LIN {X 0,Y 516.908,Z 331.095,A -85,B 0,C 180,E1 -5064.072,E2 -5064.072} C_VEL
LIN {X 0,Y 516.93,Z 331.097,A -85,B 0,C 180,E1 -5066.658,E2 -5066.658} C_VEL
LIN {X 0,Y 516.917,Z 331.093,A -85,B 0,C 180,E1 -5069.524,E2 -5069.524} C_VEL
LIN {X 0,Y 516.901,Z 331.095,A -85,B 0,C 180,E1 -5072.543,E2 -5072.543} C_VEL
LIN {X 0,Y 516.884,Z 331.1,A -85,B 0,C 180,E1 -5075.332,E2 -5075.332} C_VEL
LIN {X 0,Y 516.887,Z 331.098,A -85,B 0,C 180,E1 -5077.943,E2 -5077.943} C_VEL
LIN {X 0,Y 516.888,Z 331.102,A -85,B 0,C 180,E1 -5080.742,E2 -5080.742} C_VEL
LIN {X 0,Y 516.888,Z 331.102,A -85,B 0,C 180,E1 -5082.831,E2 -5082.831} C_VEL
LIN {X 0,Y 516.927,Z 331.093,A -85,B 0,C 180,E1 -5085.01,E2 -5085.01} C_VEL
LIN {X 0,Y 516.92,Z 331.096,A -85,B 0,C 180,E1 -5088.398,E2 -5088.398} C_VEL
LIN {X 0,Y 516.911,Z 331.249,A -85,B 0,C 180,E1 -5091.011,E2 -5091.011} C_VEL
LIN {X 0,Y 518.994,Z 341.632,A -85,B 0,C 180,E1 -5093.669,E2 -5093.669} C_VEL
LIN {X 0,Y 518.87,Z 348.689,A -85,B 0,C 180,E1 -5095.327,E2 -5095.327} C_VEL
LIN {X 0,Y 518.423,Z 362.259,A -85,B 0,C 180,E1 -5098.421,E2 -5098.421} C_VEL
LIN {X 0,Y 518.054,Z 376.981,A -85,B 0,C 180,E1 -5101.652,E2 -5101.652} C_VEL
LIN {X 0,Y 517.718,Z 390.09,A -85,B 0,C 180,E1 -5104.468,E2 -5104.468} C_VEL
LIN {X 0,Y 517.46,Z 402.865,A -85,B 0,C 180,E1 -5107.177,E2 -5107.177} C_VEL
LIN {X 0,Y 517.224,Z 417.474,A -85,B 0,C 180,E1 -5110.141,E2 -5110.141} C_VEL
LIN {X 0,Y 516.978,Z 432.958,A -85,B 0,C 180,E1 -5113.209,E2 -5113.209} C_VEL
LIN {X 0,Y 516.788,Z 447.169,A -85,B 0,C 180,E1 -5116.031,E2 -5116.031} C_VEL
LIN {X 0,Y 516.779,Z 447.609,A -85,B 0,C 180,E1 -5116.081,E2 -5116.081} C_VEL
LIN {X 0,Y 518.247,Z 458.294,A -85,B 0,C 180,E1 -5116.332,E2 -5116.332} C_VEL
LIN {X 0,Y 518.316,Z 465.73,A -85,B 0,C 180,E1 -5116.548,E2 -5116.548} C_VEL
LIN {X 0,Y 518.049,Z 479.168,A -85,B 0,C 180,E1 -5117.065,E2 -5117.065} C_VEL
LIN {X 0,Y 517.78,Z 490.854,A -85,B 0,C 180,E1 -5117.676,E2 -5117.676} C_VEL
LIN {X 0,Y 517.479,Z 502.323,A -85,B 0,C 180,E1 -5118.444,E2 -5118.444} C_VEL
LIN {X 0,Y 517.184,Z 512.955,A -85,B 0,C 180,E1 -5119.33,E2 -5119.33} C_VEL
LIN {X 0,Y 516.936,Z 521.664,A -85,B 0,C 180,E1 -5120.215,E2 -5120.215} C_VEL
LIN {X 0,Y 516.743,Z 529.713,A -85,B 0,C 180,E1 -5121.199,E2 -5121.199} C_VEL
LIN {X 0,Y 516.563,Z 537.593,A -85,B 0,C 180,E1 -5122.377,E2 -5122.377} C_VEL
LIN {X 0,Y 516.427,Z 544.854,A -85,B 0,C 180,E1 -5123.75,E2 -5123.75} C_VEL
LIN {X 0,Y 516.313,Z 549.687,A -85,B 0,C 180,E1 -5124.924,E2 -5124.924} C_VEL
LIN {X 0,Y 516.372,Z 553.401,A -85,B 0,C 180,E1 -5126.098,E2 -5126.098} C_VEL
LIN {X 0,Y 516.282,Z 555.3,A -85,B 0,C 180,E1 -5126.879,E2 -5126.879} C_VEL
LIN {X 0,Y 516.261,Z 556.732,A -85,B 0,C 180,E1 -5127.659,E2 -5127.659} C_VEL
LIN {X 0,Y 516.162,Z 558.365,A -85,B 0,C 180,E1 -5129.22,E2 -5129.22} C_VEL
LIN {X 0,Y 516.159,Z 558.585,A -85,B 0,C 180,E1 -5130,E2 -5130} C_VEL
LIN {X 0,Y 516.163,Z 558.362,A -85,B 0,C 180,E1 -5130.78,E2 -5130.78} C_VEL
LIN {X 0,Y 516.261,Z 556.725,A -85,B 0,C 180,E1 -5132.341,E2 -5132.341} C_VEL
LIN {X 0,Y 516.282,Z 555.285,A -85,B 0,C 180,E1 -5133.121,E2 -5133.121} C_VEL
LIN {X 0,Y 516.36,Z 552.268,A -85,B 0,C 180,E1 -5134.293,E2 -5134.293} C_VEL
LIN {X 0,Y 516.405,Z 548.17,A -85,B 0,C 180,E1 -5135.467,E2 -5135.467} C_VEL
LIN {X 0,Y 516.492,Z 541.976,A -85,B 0,C 180,E1 -5136.816,E2 -5136.816} C_VEL
LIN {X 0,Y 516.641,Z 534.976,A -85,B 0,C 180,E1 -5138.015,E2 -5138.015} C_VEL
LIN {X 0,Y 516.816,Z 526.424,A -85,B 0,C 180,E1 -5139.194,E2 -5139.194} C_VEL
LIN {X 0,Y 517.037,Z 517.651,A -85,B 0,C 180,E1 -5140.178,E2 -5140.178} C_VEL
LIN {X 0,Y 517.338,Z 506.848,A -85,B 0,C 180,E1 -5141.162,E2 -5141.162} C_VEL
LIN {X 0,Y 517.557,Z 495.523,A -85,B 0,C 180,E1 -5141.994,E2 -5141.994} C_VEL
LIN {X 0,Y 517.915,Z 483.454,A -85,B 0,C 180,E1 -5142.689,E2 -5142.689} C_VEL
LIN {X 0,Y 518.184,Z 469.779,A -85,B 0,C 180,E1 -5143.281,E2 -5143.281} C_VEL
LIN {X 0,Y 518.228,Z 458.613,A -85,B 0,C 180,E1 -5143.629,E2 -5143.629} C_VEL
LIN {X 0,Y 516.883,Z 448.292,A -85,B 0,C 180,E1 -5143.878,E2 -5143.878} C_VEL
LIN {X 0,Y 516.779,Z 446.249,A -85,B 0,C 180,E1 -5143.919,E2 -5143.919} C_VEL
LIN {X 0,Y 516.964,Z 430.116,A -85,B 0,C 180,E1 -5146.995,E2 -5146.995} C_VEL
LIN {X 0,Y 517.094,Z 415.047,A -85,B 0,C 180,E1 -5149.864,E2 -5149.864} C_VEL
LIN {X 0,Y 517.207,Z 399.793,A -85,B 0,C 180,E1 -5152.802,E2 -5152.802} C_VEL
LIN {X 0,Y 517.301,Z 385.694,A -85,B 0,C 180,E1 -5155.554,E2 -5155.554} C_VEL
LIN {X 0,Y 517.374,Z 371.54,A -85,B 0,C 180,E1 -5158.388,E2 -5158.388} C_VEL
LIN {X 0,Y 517.45,Z 358.184,A -85,B 0,C 180,E1 -5161.166,E2 -5161.166} C_VEL
LIN {X 0,Y 517.89,Z 341.975,A -85,B 0,C 180,E1 -5164.748,E2 -5164.748} C_VEL
LIN {X 0,Y 518.036,Z 337.974,A -85,B 0,C 180,E1 -5165.688,E2 -5165.688} C_VEL
LIN {X 0,Y 516.902,Z 331.103,A -85,B 0,C 180,E1 -5167.507,E2 -5167.507} C_VEL
LIN {X 0,Y 516.888,Z 331.103,A -85,B 0,C 180,E1 -5170.41,E2 -5170.41} C_VEL
LIN {X 0,Y 516.888,Z 331.102,A -85,B 0,C 180,E1 -5172.831,E2 -5172.831} C_VEL
LIN {X 0,Y 516.927,Z 331.095,A -85,B 0,C 180,E1 -5175.01,E2 -5175.01} C_VEL
LIN {X 0,Y 516.917,Z 331.097,A -85,B 0,C 180,E1 -5178.399,E2 -5178.399} C_VEL
LIN {X 0,Y 516.885,Z 331.101,A -85,B 0,C 180,E1 -5181.284,E2 -5181.284} C_VEL
LIN {X 0,Y 516.892,Z 331.101,A -85,B 0,C 180,E1 -5184.221,E2 -5184.221} C_VEL
LIN {X 0,Y 516.9,Z 331.1,A -85,B 0,C 180,E1 -5187.053,E2 -5187.053} C_VEL
LIN {X 0,Y 516.897,Z 331.101,A -85,B 0,C 180,E1 -5189.796,E2 -5189.796} C_VEL
LIN {X 0,Y 516.931,Z 331.095,A -85,B 0,C 180,E1 -5192.467,E2 -5192.467} C_VEL
LIN {X 0,Y 516.88,Z 331.1,A -85,B 0,C 180,E1 -5195.07,E2 -5195.07} C_VEL
LIN {X 0,Y 516.873,Z 331.102,A -85,B 0,C 180,E1 -5197.622,E2 -5197.622} C_VEL
LIN {X 0,Y 516.937,Z 331.096,A -85,B 0,C 180,E1 -5200.13,E2 -5200.13} C_VEL
LIN {X 0,Y 516.925,Z 331.098,A -85,B 0,C 180,E1 -5202.596,E2 -5202.596} C_VEL
LIN {X 0,Y 516.948,Z 331.094,A -85,B 0,C 180,E1 -5205.03,E2 -5205.03} C_VEL
LIN {X 0,Y 516.94,Z 331.279,A -85,B 0,C 180,E1 -5205.923,E2 -5205.923} C_VEL
LIN {X 0,Y 518.334,Z 336.946,A -85,B 0,C 180,E1 -5206.224,E2 -5206.224} C_VEL
LIN {X 0,Y 518.092,Z 348.48,A -85,B 0,C 180,E1 -5206.867,E2 -5206.867} C_VEL
LIN {X 0,Y 517.819,Z 359.058,A -85,B 0,C 180,E1 -5207.615,E2 -5207.615} C_VEL
LIN {X 0,Y 517.57,Z 368.563,A -85,B 0,C 180,E1 -5208.446,E2 -5208.446} C_VEL
LIN {X 0,Y 517.316,Z 377.754,A -85,B 0,C 180,E1 -5209.432,E2 -5209.432} C_VEL
LIN {X 0,Y 517.023,Z 386.607,A -85,B 0,C 180,E1 -5210.612,E2 -5210.612} C_VEL
LIN {X 0,Y 516.829,Z 393.689,A -85,B 0,C 180,E1 -5211.791,E2 -5211.791} C_VEL
LIN {X 0,Y 516.664,Z 399.315,A -85,B 0,C 180,E1 -5212.968,E2 -5212.968} C_VEL
LIN {X 0,Y 516.637,Z 403.722,A -85,B 0,C 180,E1 -5214.144,E2 -5214.144} C_VEL
LIN {X 0,Y 516.471,Z 407.079,A -85,B 0,C 180,E1 -5215.317,E2 -5215.317} C_VEL
LIN {X 0,Y 516.477,Z 408.761,A -85,B 0,C 180,E1 -5216.099,E2 -5216.099} C_VEL
LIN {X 0,Y 516.365,Z 410.885,A -85,B 0,C 180,E1 -5217.66,E2 -5217.66} C_VEL
LIN {X 0,Y 516.352,Z 411.375,A -85,B 0,C 180,E1 -5218.44,E2 -5218.44} C_VEL
LIN {X 0,Y 516.317,Z 411.149,A -85,B 0,C 180,E1 -5220,E2 -5220} C_VEL
LIN {X 0,Y 516.326,Z 410.458,A -85,B 0,C 180,E1 -5220.78,E2 -5220.78} C_VEL
LIN {X 0,Y 516.36,Z 409.365,A -85,B 0,C 180,E1 -5221.56,E2 -5221.56} C_VEL
LIN {X 0,Y 516.379,Z 407.875,A -85,B 0,C 180,E1 -5222.34,E2 -5222.34} C_VEL
LIN {X 0,Y 516.575,Z 404.822,A -85,B 0,C 180,E1 -5223.51,E2 -5223.51} C_VEL
LIN {X 0,Y 516.58,Z 400.77,A -85,B 0,C 180,E1 -5224.682,E2 -5224.682} C_VEL
LIN {X 0,Y 516.782,Z 394.527,A -85,B 0,C 180,E1 -5226.05,E2 -5226.05} C_VEL
LIN {X 0,Y 516.939,Z 387.732,A -85,B 0,C 180,E1 -5227.224,E2 -5227.224} C_VEL
LIN {X 0,Y 517.108,Z 379.256,A -85,B 0,C 180,E1 -5228.401,E2 -5228.401} C_VEL
LIN {X 0,Y 517.421,Z 370.5,A -85,B 0,C 180,E1 -5229.381,E2 -5229.381} C_VEL
LIN {X 0,Y 517.702,Z 360.917,A -85,B 0,C 180,E1 -5230.263,E2 -5230.263} C_VEL
LIN {X 0,Y 517.928,Z 350.396,A -85,B 0,C 180,E1 -5231.05,E2 -5231.05} C_VEL
LIN {X 0,Y 518.189,Z 338.681,A -85,B 0,C 180,E1 -5231.738,E2 -5231.738} C_VEL
LIN {X 0,Y 518.12,Z 335.637,A -85,B 0,C 180,E1 -5231.894,E2 -5231.894} C_VEL
LIN {X 0,Y 516.965,Z 331.093,A -85,B 0,C 180,E1 -5232.15,E2 -5232.15} C_VEL
LIN {X 0,Y 516.95,Z 331.092,A -85,B 0,C 180,E1 -5235.146,E2 -5235.146} C_VEL
LIN {X 0,Y 516.917,Z 331.092,A -85,B 0,C 180,E1 -5238.222,E2 -5238.222} C_VEL
LIN {X 0,Y 516.917,Z 331.097,A -85,B 0,C 180,E1 -5240.701,E2 -5240.701} C_VEL
LIN {X 0,Y 516.907,Z 331.098,A -85,B 0,C 180,E1 -5244.072,E2 -5244.072} C_VEL
LIN {X 0,Y 516.93,Z 331.094,A -85,B 0,C 180,E1 -5246.657,E2 -5246.657} C_VEL
LIN {X 0,Y 516.915,Z 331.099,A -85,B 0,C 180,E1 -5249.524,E2 -5249.524} C_VEL
LIN {X 0,Y 516.902,Z 331.095,A -85,B 0,C 180,E1 -5252.544,E2 -5252.544} C_VEL
LIN {X 0,Y 516.871,Z 331.101,A -85,B 0,C 180,E1 -5255.33,E2 -5255.33} C_VEL
LIN {X 0,Y 516.884,Z 331.097,A -85,B 0,C 180,E1 -5257.943,E2 -5257.943} C_VEL
LIN {X 0,Y 516.907,Z 331.097,A -85,B 0,C 180,E1 -5260.739,E2 -5260.739} C_VEL
LIN {X 0,Y 516.885,Z 331.102,A -85,B 0,C 180,E1 -5263.903,E2 -5263.903} C_VEL
LIN {X 0,Y 516.885,Z 331.099,A -85,B 0,C 180,E1 -5266.107,E2 -5266.107} C_VEL
LIN {X 0,Y 516.895,Z 331.096,A -85,B 0,C 180,E1 -5267.801,E2 -5267.801} C_VEL
LIN {X 0,Y 516.239,Z 331.179,A -85,B 0,C 180,E1 -5268.451,E2 -5268.451} C_VEL
LIN {X 0,Y 513.371,Z 331.538,A -85,B 0,C 180,E1 -5269.505,E2 -5269.505} C_VEL
LIN {X 0,Y 510.943,Z 331.839,A -85,B 0,C 180,E1 -5270.355,E2 -5270.355} C_VEL
LIN {X 0,Y 509.91,Z 331.971,A -85,B 0,C 180,E1 -5271.011,E2 -5271.011} C_VEL
LIN {X 0,Y 509.831,Z 331.975,A -85,B 0,C 180,E1 -5271.233,E2 -5271.233} C_VEL
LIN {X 0,Y 509.828,Z 331.981,A -85,B 0,C 180,E1 -5274.421,E2 -5274.421} C_VEL
LIN {X 0,Y 509.865,Z 331.973,A -85,B 0,C 180,E1 -5277.481,E2 -5277.481} C_VEL
LIN {X 0,Y 509.86,Z 331.975,A -85,B 0,C 180,E1 -5280.273,E2 -5280.273} C_VEL
LIN {X 0,Y 509.887,Z 331.972,A -85,B 0,C 180,E1 -5282.944,E2 -5282.944} C_VEL
LIN {X 0,Y 509.872,Z 331.973,A -85,B 0,C 180,E1 -5285.574,E2 -5285.574} C_VEL
LIN {X 0,Y 509.824,Z 331.978,A -85,B 0,C 180,E1 -5288.149,E2 -5288.149} C_VEL
LIN {X 0,Y 509.865,Z 331.974,A -85,B 0,C 180,E1 -5290.682,E2 -5290.682} C_VEL
LIN {X 0,Y 509.886,Z 331.968,A -85,B 0,C 180,E1 -5293.175,E2 -5293.175} C_VEL
LIN {X 0,Y 509.866,Z 331.976,A -85,B 0,C 180,E1 -5295.634,E2 -5295.634} C_VEL
LIN {X 0,Y 509.915,Z 331.968,A -85,B 0,C 180,E1 -5298.875,E2 -5298.875} C_VEL
LIN {X 0,Y 509.953,Z 331.961,A -85,B 0,C 180,E1 -5302.078,E2 -5302.078} C_VEL
LIN {X 0,Y 509.983,Z 331.963,A -85,B 0,C 180,E1 -5304.464,E2 -5304.464} C_VEL
LIN {X 0,Y 510.057,Z 331.949,A -85,B 0,C 180,E1 -5307.631,E2 -5307.631} C_VEL
LIN {X 0,Y 510.066,Z 331.946,A -85,B 0,C 180,E1 -5310.79,E2 -5310.79} C_VEL
LIN {X 0,Y 509.958,Z 331.963,A -85,B 0,C 180,E1 -5313.16,E2 -5313.16} C_VEL
LIN {X 0,Y 509.956,Z 331.961,A -85,B 0,C 180,E1 -5316.33,E2 -5316.33} C_VEL
LIN {X 0,Y 509.918,Z 331.969,A -85,B 0,C 180,E1 -5318.72,E2 -5318.72} C_VEL
LIN {X 0,Y 509.906,Z 331.97,A -85,B 0,C 180,E1 -5321.932,E2 -5321.932} C_VEL
LIN {X 0,Y 509.896,Z 331.968,A -85,B 0,C 180,E1 -5325.242,E2 -5325.242} C_VEL
LIN {X 0,Y 509.891,Z 331.97,A -85,B 0,C 180,E1 -5328.001,E2 -5328.001} C_VEL
LIN {X 0,Y 509.852,Z 331.977,A -85,B 0,C 180,E1 -5331.002,E2 -5331.002} C_VEL
LIN {X 0,Y 509.867,Z 331.976,A -85,B 0,C 180,E1 -5334.426,E2 -5334.426} C_VEL
LIN {X 0,Y 509.886,Z 331.97,A -85,B 0,C 180,E1 -5337.056,E2 -5337.056} C_VEL
LIN {X 0,Y 509.859,Z 331.977,A -85,B 0,C 180,E1 -5339.751,E2 -5339.751} C_VEL
LIN {X 0,Y 509.877,Z 331.97,A -85,B 0,C 180,E1 -5342.775,E2 -5342.775} C_VEL
LIN {X 0,Y 509.828,Z 331.979,A -85,B 0,C 180,E1 -5345.579,E2 -5345.579} C_VEL
LIN {X 0,Y 509.852,Z 331.975,A -85,B 0,C 180,E1 -5348.338,E2 -5348.338} C_VEL
LIN {X 0,Y 509.859,Z 331.973,A -85,B 0,C 180,E1 -5351.426,E2 -5351.426} C_VEL
LIN {X 0,Y 509.86,Z 331.974,A -85,B 0,C 180,E1 -5354.668,E2 -5354.668} C_VEL
LIN {X 0,Y 509.86,Z 331.974,A -85,B 0,C 180,E1 -5358.103,E2 -5358.103} C_VEL
LIN {X 0,Y 509.849,Z 331.974,A -85,B 0,C 180,E1 -5360.648,E2 -5360.648} C_VEL
LIN {X 0,Y 509.829,Z 331.976,A -85,B 0,C 180,E1 -5363.647,E2 -5363.647} C_VEL
LIN {X 0,Y 509.865,Z 331.977,A -85,B 0,C 180,E1 -5366.54,E2 -5366.54} C_VEL
LIN {X 0,Y 509.85,Z 331.974,A -85,B 0,C 180,E1 -5369.335,E2 -5369.335} C_VEL
LIN {X 0,Y 509.898,Z 331.972,A -85,B 0,C 180,E1 -5372.055,E2 -5372.055} C_VEL
LIN {X 0,Y 509.881,Z 331.97,A -85,B 0,C 180,E1 -5374.704,E2 -5374.704} C_VEL
LIN {X 0,Y 509.831,Z 331.978,A -85,B 0,C 180,E1 -5377.458,E2 -5377.458} C_VEL
LIN {X 0,Y 509.921,Z 331.963,A -85,B 0,C 180,E1 -5379.845,E2 -5379.845} C_VEL
LIN {X 0,Y 509.885,Z 331.969,A -85,B 0,C 180,E1 -5383.175,E2 -5383.175} C_VEL
LIN {X 0,Y 509.87,Z 331.974,A -85,B 0,C 180,E1 -5385.634,E2 -5385.634} C_VEL
LIN {X 0,Y 509.919,Z 331.966,A -85,B 0,C 180,E1 -5388.875,E2 -5388.875} C_VEL
LIN {X 0,Y 509.958,Z 331.96,A -85,B 0,C 180,E1 -5392.079,E2 -5392.079} C_VEL
LIN {X 0,Y 509.987,Z 331.959,A -85,B 0,C 180,E1 -5394.464,E2 -5394.464} C_VEL
LIN {X 0,Y 510.058,Z 331.946,A -85,B 0,C 180,E1 -5397.631,E2 -5397.631} C_VEL
LIN {X 0,Y 510.07,Z 331.947,A -85,B 0,C 180,E1 -5400.79,E2 -5400.79} C_VEL
LIN {X 0,Y 509.96,Z 331.961,A -85,B 0,C 180,E1 -5403.16,E2 -5403.16} C_VEL
LIN {X 0,Y 509.959,Z 331.961,A -85,B 0,C 180,E1 -5406.33,E2 -5406.33} C_VEL
LIN {X 0,Y 509.911,Z 331.97,A -85,B 0,C 180,E1 -5408.72,E2 -5408.72} C_VEL
LIN {X 0,Y 509.911,Z 331.966,A -85,B 0,C 180,E1 -5411.932,E2 -5411.932} C_VEL
LIN {X 0,Y 509.9,Z 331.966,A -85,B 0,C 180,E1 -5415.242,E2 -5415.242} C_VEL
LIN {X 0,Y 509.895,Z 331.973,A -85,B 0,C 180,E1 -5418.001,E2 -5418.001} C_VEL
LIN {X 0,Y 509.857,Z 331.975,A -85,B 0,C 180,E1 -5421.002,E2 -5421.002} C_VEL
LIN {X 0,Y 509.87,Z 331.973,A -85,B 0,C 180,E1 -5424.426,E2 -5424.426} C_VEL
LIN {X 0,Y 509.889,Z 331.972,A -85,B 0,C 180,E1 -5427.056,E2 -5427.056} C_VEL
LIN {X 0,Y 509.863,Z 331.973,A -85,B 0,C 180,E1 -5429.751,E2 -5429.751} C_VEL
LIN {X 0,Y 509.878,Z 331.969,A -85,B 0,C 180,E1 -5432.774,E2 -5432.774} C_VEL
LIN {X 0,Y 509.844,Z 331.98,A -85,B 0,C 180,E1 -5435.58,E2 -5435.58} C_VEL
LIN {X 0,Y 509.856,Z 331.973,A -85,B 0,C 180,E1 -5438.338,E2 -5438.338} C_VEL
LIN {X 0,Y 509.86,Z 331.974,A -85,B 0,C 180,E1 -5441.425,E2 -5441.425} C_VEL
LIN {X 0,Y 509.862,Z 331.977,A -85,B 0,C 180,E1 -5444.668,E2 -5444.668} C_VEL
LIN {X 0,Y 509.864,Z 331.977,A -85,B 0,C 180,E1 -5448.103,E2 -5448.103} C_VEL
LIN {X 0,Y 509.866,Z 332.045,A -85,B 0,C 180,E1 -5450.713,E2 -5450.713} C_VEL
LIN {X 0,Y 511.894,Z 342.129,A -85,B 0,C 180,E1 -5453.341,E2 -5453.341} C_VEL
LIN {X 0,Y 512.14,Z 346.602,A -85,B 0,C 180,E1 -5454.431,E2 -5454.431} C_VEL
LIN {X 0,Y 511.556,Z 361.233,A -85,B 0,C 180,E1 -5457.834,E2 -5457.834} C_VEL
LIN {X 0,Y 511.098,Z 376.354,A -85,B 0,C 180,E1 -5461.231,E2 -5461.231} C_VEL
LIN {X 0,Y 510.732,Z 389.473,A -85,B 0,C 180,E1 -5464.093,E2 -5464.093} C_VEL
LIN {X 0,Y 510.455,Z 402.496,A -85,B 0,C 180,E1 -5466.897,E2 -5466.897} C_VEL
LIN {X 0,Y 510.221,Z 414.988,A -85,B 0,C 180,E1 -5469.499,E2 -5469.499} C_VEL
LIN {X 0,Y 509.975,Z 431.227,A -85,B 0,C 180,E1 -5472.765,E2 -5472.765} C_VEL
LIN {X 0,Y 509.729,Z 445.315,A -85,B 0,C 180,E1 -5475.63,E2 -5475.63} C_VEL
LIN {X 0,Y 509.722,Z 446.55,A -85,B 0,C 180,E1 -5475.885,E2 -5475.885} C_VEL
LIN {X 0,Y 510.992,Z 457.207,A -85,B 0,C 180,E1 -5476.136,E2 -5476.136} C_VEL
LIN {X 0,Y 511.46,Z 462.268,A -85,B 0,C 180,E1 -5476.288,E2 -5476.288} C_VEL
LIN {X 0,Y 511.141,Z 474.694,A -85,B 0,C 180,E1 -5476.735,E2 -5476.735} C_VEL
LIN {X 0,Y 510.822,Z 487.491,A -85,B 0,C 180,E1 -5477.37,E2 -5477.37} C_VEL
LIN {X 0,Y 510.544,Z 498.597,A -85,B 0,C 180,E1 -5478.083,E2 -5478.083} C_VEL
LIN {X 0,Y 510.197,Z 509.748,A -85,B 0,C 180,E1 -5478.981,E2 -5478.981} C_VEL
LIN {X 0,Y 509.873,Z 520.644,A -85,B 0,C 180,E1 -5480.078,E2 -5480.078} C_VEL
LIN {X 0,Y 509.681,Z 528.707,A -85,B 0,C 180,E1 -5481.076,E2 -5481.076} C_VEL
LIN {X 0,Y 509.514,Z 536.607,A -85,B 0,C 180,E1 -5482.271,E2 -5482.271} C_VEL
LIN {X 0,Y 509.346,Z 543.872,A -85,B 0,C 180,E1 -5483.662,E2 -5483.662} C_VEL
LIN {X 0,Y 509.275,Z 548.715,A -85,B 0,C 180,E1 -5484.854,E2 -5484.854} C_VEL
LIN {X 0,Y 509.336,Z 552.432,A -85,B 0,C 180,E1 -5486.044,E2 -5486.044} C_VEL
LIN {X 0,Y 509.237,Z 554.326,A -85,B 0,C 180,E1 -5486.835,E2 -5486.835} C_VEL
LIN {X 0,Y 509.217,Z 555.758,A -85,B 0,C 180,E1 -5487.627,E2 -5487.627} C_VEL
LIN {X 0,Y 509.129,Z 557.385,A -85,B 0,C 180,E1 -5489.209,E2 -5489.209} C_VEL
LIN {X 0,Y 509.149,Z 557.596,A -85,B 0,C 180,E1 -5490,E2 -5490} C_VEL
LIN {X 0,Y 509.156,Z 557.366,A -85,B 0,C 180,E1 -5490.791,E2 -5490.791} C_VEL
LIN {X 0,Y 509.223,Z 555.705,A -85,B 0,C 180,E1 -5492.373,E2 -5492.373} C_VEL
LIN {X 0,Y 509.245,Z 554.244,A -85,B 0,C 180,E1 -5493.164,E2 -5493.164} C_VEL
LIN {X 0,Y 509.3,Z 551.196,A -85,B 0,C 180,E1 -5494.353,E2 -5494.353} C_VEL
LIN {X 0,Y 509.358,Z 547.068,A -85,B 0,C 180,E1 -5495.543,E2 -5495.543} C_VEL
LIN {X 0,Y 509.421,Z 541.059,A -85,B 0,C 180,E1 -5496.868,E2 -5496.868} C_VEL
LIN {X 0,Y 509.573,Z 533.79,A -85,B 0,C 180,E1 -5498.127,E2 -5498.127} C_VEL
LIN {X 0,Y 509.77,Z 525.183,A -85,B 0,C 180,E1 -5499.323,E2 -5499.323} C_VEL
LIN {X 0,Y 510.028,Z 515.354,A -85,B 0,C 180,E1 -5500.42,E2 -5500.42} C_VEL
LIN {X 0,Y 510.324,Z 504.283,A -85,B 0,C 180,E1 -5501.418,E2 -5501.418} C_VEL
LIN {X 0,Y 510.59,Z 492.953,A -85,B 0,C 180,E1 -5502.236,E2 -5502.236} C_VEL
LIN {X 0,Y 510.912,Z 480.946,A -85,B 0,C 180,E1 -5502.917,E2 -5502.917} C_VEL
LIN {X 0,Y 511.194,Z 468.245,A -85,B 0,C 180,E1 -5503.466,E2 -5503.466} C_VEL
LIN {X 0,Y 511.23,Z 459.231,A -85,B 0,C 180,E1 -5503.756,E2 -5503.756} C_VEL
LIN {X 0,Y 509.951,Z 448.798,A -85,B 0,C 180,E1 -5504.033,E2 -5504.033} C_VEL
LIN {X 0,Y 509.728,Z 444.968,A -85,B 0,C 180,E1 -5504.115,E2 -5504.115} C_VEL
LIN {X 0,Y 509.885,Z 428.825,A -85,B 0,C 180,E1 -5507.238,E2 -5507.238} C_VEL
LIN {X 0,Y 510.064,Z 412.232,A -85,B 0,C 180,E1 -5510.454,E2 -5510.454} C_VEL
LIN {X 0,Y 510.181,Z 395.371,A -85,B 0,C 180,E1 -5513.762,E2 -5513.762} C_VEL
LIN {X 0,Y 510.301,Z 380.687,A -85,B 0,C 180,E1 -5516.708,E2 -5516.708} C_VEL
LIN {X 0,Y 510.375,Z 365.654,A -85,B 0,C 180,E1 -5519.827,E2 -5519.827} C_VEL
LIN {X 0,Y 510.537,Z 353.484,A -85,B 0,C 180,E1 -5522.471,E2 -5522.471} C_VEL
LIN {X 0,Y 511.088,Z 340.285,A -85,B 0,C 180,E1 -5525.526,E2 -5525.526} C_VEL
LIN {X 0,Y 510.634,Z 336.003,A -85,B 0,C 180,E1 -5526.628,E2 -5526.628} C_VEL
LIN {X 0,Y 509.85,Z 331.981,A -85,B 0,C 180,E1 -5527.774,E2 -5527.774} C_VEL
LIN {X 0,Y 509.843,Z 331.979,A -85,B 0,C 180,E1 -5530.698,E2 -5530.698} C_VEL
LIN {X 0,Y 509.824,Z 331.981,A -85,B 0,C 180,E1 -5533.572,E2 -5533.572} C_VEL
LIN {X 0,Y 509.823,Z 331.979,A -85,B 0,C 180,E1 -5536.428,E2 -5536.428} C_VEL
LIN {X 0,Y 509.842,Z 331.977,A -85,B 0,C 180,E1 -5539.302,E2 -5539.302} C_VEL
LIN {X 0,Y 509.855,Z 331.976,A -85,B 0,C 180,E1 -5541.786,E2 -5541.786} C_VEL
LIN {X 0,Y 509.847,Z 331.978,A -85,B 0,C 180,E1 -5544.623,E2 -5544.623} C_VEL
LIN {X 0,Y 509.866,Z 331.975,A -85,B 0,C 180,E1 -5547.481,E2 -5547.481} C_VEL
LIN {X 0,Y 509.863,Z 331.975,A -85,B 0,C 180,E1 -5550.274,E2 -5550.274} C_VEL
LIN {X 0,Y 509.889,Z 331.973,A -85,B 0,C 180,E1 -5552.944,E2 -5552.944} C_VEL
LIN {X 0,Y 509.856,Z 331.978,A -85,B 0,C 180,E1 -5555.573,E2 -5555.573} C_VEL
LIN {X 0,Y 509.827,Z 331.982,A -85,B 0,C 180,E1 -5558.149,E2 -5558.149} C_VEL
LIN {X 0,Y 509.868,Z 331.976,A -85,B 0,C 180,E1 -5560.682,E2 -5560.682} C_VEL
LIN {X 0,Y 509.885,Z 331.973,A -85,B 0,C 180,E1 -5563.175,E2 -5563.175} C_VEL
LIN {X 0,Y 509.886,Z 332.091,A -85,B 0,C 180,E1 -5565.736,E2 -5565.736} C_VEL
LIN {X 0,Y 511.443,Z 338.53,A -85,B 0,C 180,E1 -5566.085,E2 -5566.085} C_VEL
LIN {X 0,Y 511.163,Z 350.716,A -85,B 0,C 180,E1 -5566.786,E2 -5566.786} C_VEL
LIN {X 0,Y 510.87,Z 362.015,A -85,B 0,C 180,E1 -5567.621,E2 -5567.621} C_VEL
LIN {X 0,Y 510.599,Z 371.402,A -85,B 0,C 180,E1 -5568.487,E2 -5568.487} C_VEL
LIN {X 0,Y 510.351,Z 380.243,A -85,B 0,C 180,E1 -5569.487,E2 -5569.487} C_VEL
LIN {X 0,Y 510.069,Z 388.834,A -85,B 0,C 180,E1 -5570.683,E2 -5570.683} C_VEL
LIN {X 0,Y 509.842,Z 395.671,A -85,B 0,C 180,E1 -5571.877,E2 -5571.877} C_VEL
LIN {X 0,Y 509.648,Z 401.468,A -85,B 0,C 180,E1 -5573.159,E2 -5573.159} C_VEL
LIN {X 0,Y 509.563,Z 405.95,A -85,B 0,C 180,E1 -5574.46,E2 -5574.46} C_VEL
LIN {X 0,Y 509.464,Z 408.083,A -85,B 0,C 180,E1 -5575.252,E2 -5575.252} C_VEL
LIN {X 0,Y 509.461,Z 409.77,A -85,B 0,C 180,E1 -5576.045,E2 -5576.045} C_VEL
LIN {X 0,Y 509.344,Z 411.897,A -85,B 0,C 180,E1 -5577.627,E2 -5577.627} C_VEL
LIN {X 0,Y 509.341,Z 412.386,A -85,B 0,C 180,E1 -5578.419,E2 -5578.419} C_VEL
LIN {X 0,Y 509.295,Z 412.157,A -85,B 0,C 180,E1 -5580,E2 -5580} C_VEL
LIN {X 0,Y 509.349,Z 410.365,A -85,B 0,C 180,E1 -5581.581,E2 -5581.581} C_VEL
LIN {X 0,Y 509.356,Z 408.871,A -85,B 0,C 180,E1 -5582.372,E2 -5582.372} C_VEL
LIN {X 0,Y 509.571,Z 405.805,A -85,B 0,C 180,E1 -5583.558,E2 -5583.558} C_VEL
LIN {X 0,Y 509.57,Z 401.739,A -85,B 0,C 180,E1 -5584.747,E2 -5584.747} C_VEL
LIN {X 0,Y 509.789,Z 395.475,A -85,B 0,C 180,E1 -5586.133,E2 -5586.133} C_VEL
LIN {X 0,Y 509.968,Z 388.665,A -85,B 0,C 180,E1 -5587.324,E2 -5587.324} C_VEL
LIN {X 0,Y 510.155,Z 380.169,A -85,B 0,C 180,E1 -5588.516,E2 -5588.516} C_VEL
LIN {X 0,Y 510.489,Z 371.4,A -85,B 0,C 180,E1 -5589.509,E2 -5589.509} C_VEL
LIN {X 0,Y 510.792,Z 361.804,A -85,B 0,C 180,E1 -5590.404,E2 -5590.404} C_VEL
LIN {X 0,Y 511.02,Z 351.287,A -85,B 0,C 180,E1 -5591.201,E2 -5591.201} C_VEL
LIN {X 0,Y 511.295,Z 339.58,A -85,B 0,C 180,E1 -5591.899,E2 -5591.899} C_VEL
LIN {X 0,Y 511.056,Z 336.268,A -85,B 0,C 180,E1 -5592.076,E2 -5592.076} C_VEL
LIN {X 0,Y 509.901,Z 331.972,A -85,B 0,C 180,E1 -5592.336,E2 -5592.336} C_VEL
LIN {X 0,Y 509.899,Z 331.971,A -85,B 0,C 180,E1 -5595.242,E2 -5595.242} C_VEL
LIN {X 0,Y 509.862,Z 331.971,A -85,B 0,C 180,E1 -5598.484,E2 -5598.484} C_VEL
LIN {X 0,Y 509.854,Z 331.978,A -85,B 0,C 180,E1 -5601.001,E2 -5601.001} C_VEL
LIN {X 0,Y 509.868,Z 331.976,A -85,B 0,C 180,E1 -5604.426,E2 -5604.426} C_VEL
LIN {X 0,Y 509.889,Z 331.969,A -85,B 0,C 180,E1 -5607.055,E2 -5607.055} C_VEL
LIN {X 0,Y 509.861,Z 331.977,A -85,B 0,C 180,E1 -5609.751,E2 -5609.751} C_VEL
LIN {X 0,Y 509.878,Z 331.971,A -85,B 0,C 180,E1 -5612.774,E2 -5612.774} C_VEL
LIN {X 0,Y 509.83,Z 331.976,A -85,B 0,C 180,E1 -5615.578,E2 -5615.578} C_VEL
LIN {X 0,Y 509.855,Z 331.976,A -85,B 0,C 180,E1 -5618.338,E2 -5618.338} C_VEL
LIN {X 0,Y 509.869,Z 331.972,A -85,B 0,C 180,E1 -5621.424,E2 -5621.424} C_VEL
LIN {X 0,Y 509.859,Z 331.973,A -85,B 0,C 180,E1 -5624.668,E2 -5624.668} C_VEL
LIN {X 0,Y 509.863,Z 331.973,A -85,B 0,C 180,E1 -5628.102,E2 -5628.102} C_VEL
LIN {X 0,Y 509.831,Z 331.975,A -85,B 0,C 180,E1 -5631.233,E2 -5631.233} C_VEL
LIN {X 0,Y 509.171,Z 332.058,A -85,B 0,C 180,E1 -5631.892,E2 -5631.892} C_VEL
LIN {X 0,Y 506.297,Z 332.419,A -85,B 0,C 180,E1 -5632.961,E2 -5632.961} C_VEL
LIN {X 0,Y 503.874,Z 332.719,A -85,B 0,C 180,E1 -5633.823,E2 -5633.823} C_VEL
LIN {X 0,Y 502.851,Z 332.851,A -85,B 0,C 180,E1 -5634.488,E2 -5634.488} C_VEL
LIN {X 0,Y 502.778,Z 332.854,A -85,B 0,C 180,E1 -5634.713,E2 -5634.713} C_VEL
LIN {X 0,Y 502.834,Z 332.848,A -85,B 0,C 180,E1 -5636.993,E2 -5636.993} C_VEL
LIN {X 0,Y 502.816,Z 332.854,A -85,B 0,C 180,E1 -5640.065,E2 -5640.065} C_VEL
LIN {X 0,Y 502.835,Z 332.848,A -85,B 0,C 180,E1 -5642.533,E2 -5642.533} C_VEL
LIN {X 0,Y 502.831,Z 332.852,A -85,B 0,C 180,E1 -5645.298,E2 -5645.298} C_VEL
LIN {X 0,Y 502.795,Z 332.852,A -85,B 0,C 180,E1 -5647.827,E2 -5647.827} C_VEL
LIN {X 0,Y 502.827,Z 332.855,A -85,B 0,C 180,E1 -5650.4,E2 -5650.4} C_VEL
LIN {X 0,Y 502.836,Z 332.847,A -85,B 0,C 180,E1 -5652.932,E2 -5652.932} C_VEL
LIN {X 0,Y 502.847,Z 332.849,A -85,B 0,C 180,E1 -5655.429,E2 -5655.429} C_VEL
LIN {X 0,Y 502.879,Z 332.844,A -85,B 0,C 180,E1 -5658.717,E2 -5658.717} C_VEL
LIN {X 0,Y 502.903,Z 332.84,A -85,B 0,C 180,E1 -5661.967,E2 -5661.967} C_VEL
LIN {X 0,Y 502.937,Z 332.84,A -85,B 0,C 180,E1 -5664.387,E2 -5664.387} C_VEL
LIN {X 0,Y 503.027,Z 332.824,A -85,B 0,C 180,E1 -5667.598,E2 -5667.598} C_VEL
LIN {X 0,Y 503.029,Z 332.828,A -85,B 0,C 180,E1 -5670,E2 -5670} C_VEL
LIN {X 0,Y 503.028,Z 332.824,A -85,B 0,C 180,E1 -5672.402,E2 -5672.402} C_VEL
LIN {X 0,Y 502.936,Z 332.838,A -85,B 0,C 180,E1 -5675.614,E2 -5675.614} C_VEL
LIN {X 0,Y 502.904,Z 332.84,A -85,B 0,C 180,E1 -5678.033,E2 -5678.033} C_VEL
LIN {X 0,Y 502.88,Z 332.842,A -85,B 0,C 180,E1 -5681.283,E2 -5681.283} C_VEL
LIN {X 0,Y 502.847,Z 332.846,A -85,B 0,C 180,E1 -5684.571,E2 -5684.571} C_VEL
LIN {X 0,Y 502.864,Z 332.846,A -85,B 0,C 180,E1 -5687.907,E2 -5687.907} C_VEL
LIN {X 0,Y 502.83,Z 332.849,A -85,B 0,C 180,E1 -5690.536,E2 -5690.536} C_VEL
LIN {X 0,Y 502.793,Z 332.858,A -85,B 0,C 180,E1 -5693.041,E2 -5693.041} C_VEL
LIN {X 0,Y 502.842,Z 332.847,A -85,B 0,C 180,E1 -5695.676,E2 -5695.676} C_VEL
LIN {X 0,Y 502.842,Z 332.85,A -85,B 0,C 180,E1 -5698.373,E2 -5698.373} C_VEL
LIN {X 0,Y 502.796,Z 332.856,A -85,B 0,C 180,E1 -5701.499,E2 -5701.499} C_VEL
LIN {X 0,Y 502.806,Z 332.851,A -85,B 0,C 180,E1 -5703.994,E2 -5703.994} C_VEL
LIN {X 0,Y 502.78,Z 332.86,A -85,B 0,C 180,E1 -5707.178,E2 -5707.178} C_VEL
LIN {X 0,Y 502.79,Z 332.854,A -85,B 0,C 180,E1 -5710.015,E2 -5710.015} C_VEL
LIN {X 0,Y 502.833,Z 332.852,A -85,B 0,C 180,E1 -5712.203,E2 -5712.203} C_VEL
LIN {X 0,Y 502.804,Z 332.854,A -85,B 0,C 180,E1 -5715.468,E2 -5715.468} C_VEL
LIN {X 0,Y 502.823,Z 332.85,A -85,B 0,C 180,E1 -5718.934,E2 -5718.934} C_VEL
LIN {X 0,Y 502.796,Z 332.851,A -85,B 0,C 180,E1 -5722.046,E2 -5722.046} C_VEL
LIN {X 0,Y 502.806,Z 332.855,A -85,B 0,C 180,E1 -5725.035,E2 -5725.035} C_VEL
LIN {X 0,Y 502.788,Z 332.856,A -85,B 0,C 180,E1 -5727.916,E2 -5727.916} C_VEL
LIN {X 0,Y 502.829,Z 332.85,A -85,B 0,C 180,E1 -5730.713,E2 -5730.713} C_VEL
LIN {X 0,Y 502.867,Z 332.849,A -85,B 0,C 180,E1 -5733.44,E2 -5733.44} C_VEL
LIN {X 0,Y 502.79,Z 332.853,A -85,B 0,C 180,E1 -5736.086,E2 -5736.086} C_VEL
LIN {X 0,Y 502.788,Z 332.857,A -85,B 0,C 180,E1 -5738.689,E2 -5738.689} C_VEL
LIN {X 0,Y 502.831,Z 332.848,A -85,B 0,C 180,E1 -5741.248,E2 -5741.248} C_VEL
LIN {X 0,Y 502.825,Z 332.85,A -85,B 0,C 180,E1 -5743.767,E2 -5743.767} C_VEL
LIN {X 0,Y 502.837,Z 332.852,A -85,B 0,C 180,E1 -5746.255,E2 -5746.255} C_VEL
LIN {X 0,Y 502.883,Z 332.842,A -85,B 0,C 180,E1 -5748.717,E2 -5748.717} C_VEL
LIN {X 0,Y 502.908,Z 332.839,A -85,B 0,C 180,E1 -5751.967,E2 -5751.967} C_VEL
LIN {X 0,Y 502.943,Z 332.836,A -85,B 0,C 180,E1 -5754.387,E2 -5754.387} C_VEL
LIN {X 0,Y 503.028,Z 332.822,A -85,B 0,C 180,E1 -5757.598,E2 -5757.598} C_VEL
LIN {X 0,Y 503.034,Z 332.826,A -85,B 0,C 180,E1 -5760,E2 -5760} C_VEL
LIN {X 0,Y 503.031,Z 332.825,A -85,B 0,C 180,E1 -5762.402,E2 -5762.402} C_VEL
LIN {X 0,Y 502.937,Z 332.839,A -85,B 0,C 180,E1 -5765.614,E2 -5765.614} C_VEL
LIN {X 0,Y 502.887,Z 332.842,A -85,B 0,C 180,E1 -5768.034,E2 -5768.034} C_VEL
LIN {X 0,Y 502.883,Z 332.843,A -85,B 0,C 180,E1 -5771.283,E2 -5771.283} C_VEL
LIN {X 0,Y 502.851,Z 332.848,A -85,B 0,C 180,E1 -5774.571,E2 -5774.571} C_VEL
LIN {X 0,Y 502.868,Z 332.849,A -85,B 0,C 180,E1 -5777.907,E2 -5777.907} C_VEL
LIN {X 0,Y 502.835,Z 332.848,A -85,B 0,C 180,E1 -5780.536,E2 -5780.536} C_VEL
LIN {X 0,Y 502.797,Z 332.856,A -85,B 0,C 180,E1 -5783.041,E2 -5783.041} C_VEL
LIN {X 0,Y 502.845,Z 332.847,A -85,B 0,C 180,E1 -5785.675,E2 -5785.675} C_VEL
LIN {X 0,Y 502.845,Z 332.852,A -85,B 0,C 180,E1 -5788.373,E2 -5788.373} C_VEL
LIN {X 0,Y 502.798,Z 332.852,A -85,B 0,C 180,E1 -5791.499,E2 -5791.499} C_VEL
LIN {X 0,Y 502.81,Z 332.851,A -85,B 0,C 180,E1 -5794.444,E2 -5794.444} C_VEL
LIN {X 0,Y 502.786,Z 332.857,A -85,B 0,C 180,E1 -5797.178,E2 -5797.178} C_VEL
LIN {X 0,Y 502.793,Z 332.853,A -85,B 0,C 180,E1 -5800.015,E2 -5800.015} C_VEL
LIN {X 0,Y 502.807,Z 332.854,A -85,B 0,C 180,E1 -5802.199,E2 -5802.199} C_VEL
LIN {X 0,Y 502.806,Z 332.852,A -85,B 0,C 180,E1 -5805.468,E2 -5805.468} C_VEL
LIN {X 0,Y 502.834,Z 332.852,A -85,B 0,C 180,E1 -5807.864,E2 -5807.864} C_VEL
LIN {X 0,Y 502.825,Z 333.026,A -85,B 0,C 180,E1 -5810.461,E2 -5810.461} C_VEL
LIN {X 0,Y 504.961,Z 343.532,A -85,B 0,C 180,E1 -5813.239,E2 -5813.239} C_VEL
LIN {X 0,Y 505.226,Z 347.589,A -85,B 0,C 180,E1 -5814.25,E2 -5814.25} C_VEL
LIN {X 0,Y 504.632,Z 360.686,A -85,B 0,C 180,E1 -5817.338,E2 -5817.338} C_VEL
LIN {X 0,Y 504.164,Z 373.742,A -85,B 0,C 180,E1 -5820.339,E2 -5820.339} C_VEL
LIN {X 0,Y 503.844,Z 387.854,A -85,B 0,C 180,E1 -5823.489,E2 -5823.489} C_VEL
LIN {X 0,Y 503.443,Z 401.886,A -85,B 0,C 180,E1 -5826.555,E2 -5826.555} C_VEL
LIN {X 0,Y 503.139,Z 416.038,A -85,B 0,C 180,E1 -5829.561,E2 -5829.561} C_VEL
LIN {X 0,Y 502.913,Z 431.546,A -85,B 0,C 180,E1 -5832.725,E2 -5832.725} C_VEL
LIN {X 0,Y 502.648,Z 445.682,A -85,B 0,C 180,E1 -5835.682,E2 -5835.682} C_VEL
LIN {X 0,Y 503.941,Z 457.493,A -85,B 0,C 180,E1 -5835.977,E2 -5835.977} C_VEL
LIN {X 0,Y 504.528,Z 462.007,A -85,B 0,C 180,E1 -5836.122,E2 -5836.122} C_VEL
LIN {X 0,Y 504.166,Z 474.76,A -85,B 0,C 180,E1 -5836.6,E2 -5836.6} C_VEL
LIN {X 0,Y 503.808,Z 486.643,A -85,B 0,C 180,E1 -5837.205,E2 -5837.205} C_VEL
LIN {X 0,Y 503.502,Z 498.931,A -85,B 0,C 180,E1 -5838.016,E2 -5838.016} C_VEL
LIN {X 0,Y 503.115,Z 509.807,A -85,B 0,C 180,E1 -5838.926,E2 -5838.926} C_VEL
LIN {X 0,Y 502.802,Z 519.622,A -85,B 0,C 180,E1 -5839.937,E2 -5839.937} C_VEL
LIN {X 0,Y 502.602,Z 527.698,A -85,B 0,C 180,E1 -5840.949,E2 -5840.949} C_VEL
LIN {X 0,Y 502.433,Z 535.615,A -85,B 0,C 180,E1 -5842.161,E2 -5842.161} C_VEL
LIN {X 0,Y 502.275,Z 542.889,A -85,B 0,C 180,E1 -5843.573,E2 -5843.573} C_VEL
LIN {X 0,Y 502.236,Z 547.741,A -85,B 0,C 180,E1 -5844.781,E2 -5844.781} C_VEL
LIN {X 0,Y 502.276,Z 551.458,A -85,B 0,C 180,E1 -5845.988,E2 -5845.988} C_VEL
LIN {X 0,Y 502.192,Z 553.352,A -85,B 0,C 180,E1 -5846.791,E2 -5846.791} C_VEL
LIN {X 0,Y 502.173,Z 554.784,A -85,B 0,C 180,E1 -5847.594,E2 -5847.594} C_VEL
LIN {X 0,Y 502.12,Z 555.793,A -85,B 0,C 180,E1 -5848.396,E2 -5848.396} C_VEL
LIN {X 0,Y 502.096,Z 556.401,A -85,B 0,C 180,E1 -5849.198,E2 -5849.198} C_VEL
LIN {X 0,Y 502.138,Z 556.608,A -85,B 0,C 180,E1 -5850,E2 -5850} C_VEL
LIN {X 0,Y 502.147,Z 556.371,A -85,B 0,C 180,E1 -5850.802,E2 -5850.802} C_VEL
LIN {X 0,Y 502.185,Z 554.68,A -85,B 0,C 180,E1 -5852.406,E2 -5852.406} C_VEL
LIN {X 0,Y 502.207,Z 553.202,A -85,B 0,C 180,E1 -5853.209,E2 -5853.209} C_VEL
LIN {X 0,Y 502.248,Z 550.125,A -85,B 0,C 180,E1 -5854.414,E2 -5854.414} C_VEL
LIN {X 0,Y 502.305,Z 545.966,A -85,B 0,C 180,E1 -5855.621,E2 -5855.621} C_VEL
LIN {X 0,Y 502.359,Z 539.675,A -85,B 0,C 180,E1 -5857.011,E2 -5857.011} C_VEL
LIN {X 0,Y 502.499,Z 532.599,A -85,B 0,C 180,E1 -5858.242,E2 -5858.242} C_VEL
LIN {X 0,Y 502.719,Z 523.939,A -85,B 0,C 180,E1 -5859.455,E2 -5859.455} C_VEL
LIN {X 0,Y 502.932,Z 514.045,A -85,B 0,C 180,E1 -5860.568,E2 -5860.568} C_VEL
LIN {X 0,Y 503.327,Z 502.929,A -85,B 0,C 180,E1 -5861.579,E2 -5861.579} C_VEL
LIN {X 0,Y 503.595,Z 491.678,A -85,B 0,C 180,E1 -5862.399,E2 -5862.399} C_VEL
LIN {X 0,Y 503.93,Z 479.464,A -85,B 0,C 180,E1 -5863.099,E2 -5863.099} C_VEL
LIN {X 0,Y 504.269,Z 466.723,A -85,B 0,C 180,E1 -5863.654,E2 -5863.654} C_VEL
LIN {X 0,Y 504.232,Z 459.901,A -85,B 0,C 180,E1 -5863.886,E2 -5863.886} C_VEL
LIN {X 0,Y 503.048,Z 449.786,A -85,B 0,C 180,E1 -5864.178,E2 -5864.178} C_VEL
LIN {X 0,Y 502.621,Z 443.675,A -85,B 0,C 180,E1 -5864.319,E2 -5864.319} C_VEL
LIN {X 0,Y 502.801,Z 429.654,A -85,B 0,C 180,E1 -5867.07,E2 -5867.07} C_VEL
LIN {X 0,Y 502.958,Z 413.604,A -85,B 0,C 180,E1 -5870.233,E2 -5870.233} C_VEL
LIN {X 0,Y 503.095,Z 397.411,A -85,B 0,C 180,E1 -5873.462,E2 -5873.462} C_VEL
LIN {X 0,Y 503.213,Z 383.364,A -85,B 0,C 180,E1 -5876.323,E2 -5876.323} C_VEL
LIN {X 0,Y 503.319,Z 369.421,A -85,B 0,C 180,E1 -5879.256,E2 -5879.256} C_VEL
LIN {X 0,Y 503.528,Z 356.786,A -85,B 0,C 180,E1 -5882.032,E2 -5882.032} C_VEL
LIN {X 0,Y 504.101,Z 342.64,A -85,B 0,C 180,E1 -5885.351,E2 -5885.351} C_VEL
LIN {X 0,Y 503.913,Z 338.571,A -85,B 0,C 180,E1 -5886.398,E2 -5886.398} C_VEL
LIN {X 0,Y 502.826,Z 332.856,A -85,B 0,C 180,E1 -5888.051,E2 -5888.051} C_VEL
LIN {X 0,Y 502.824,Z 332.853,A -85,B 0,C 180,E1 -5891.066,E2 -5891.066} C_VEL
LIN {X 0,Y 502.805,Z 332.857,A -85,B 0,C 180,E1 -5894.532,E2 -5894.532} C_VEL
LIN {X 0,Y 502.799,Z 332.854,A -85,B 0,C 180,E1 -5897.861,E2 -5897.861} C_VEL
LIN {X 0,Y 502.805,Z 332.853,A -85,B 0,C 180,E1 -5901.024,E2 -5901.024} C_VEL
LIN {X 0,Y 502.787,Z 332.858,A -85,B 0,C 180,E1 -5904.168,E2 -5904.168} C_VEL
LIN {X 0,Y 502.837,Z 332.852,A -85,B 0,C 180,E1 -5906.993,E2 -5906.993} C_VEL
LIN {X 0,Y 502.819,Z 332.853,A -85,B 0,C 180,E1 -5910.065,E2 -5910.065} C_VEL
LIN {X 0,Y 502.837,Z 332.851,A -85,B 0,C 180,E1 -5912.533,E2 -5912.533} C_VEL
LIN {X 0,Y 502.808,Z 332.855,A -85,B 0,C 180,E1 -5915.305,E2 -5915.305} C_VEL
LIN {X 0,Y 502.785,Z 332.857,A -85,B 0,C 180,E1 -5917.826,E2 -5917.826} C_VEL
LIN {X 0,Y 502.829,Z 332.852,A -85,B 0,C 180,E1 -5920.4,E2 -5920.4} C_VEL
LIN {X 0,Y 502.833,Z 332.852,A -85,B 0,C 180,E1 -5922.931,E2 -5922.931} C_VEL
LIN {X 0,Y 502.836,Z 332.943,A -85,B 0,C 180,E1 -5925.545,E2 -5925.545} C_VEL
LIN {X 0,Y 504.542,Z 339.126,A -85,B 0,C 180,E1 -5925.891,E2 -5925.891} C_VEL
LIN {X 0,Y 504.306,Z 351.408,A -85,B 0,C 180,E1 -5926.604,E2 -5926.604} C_VEL
LIN {X 0,Y 503.997,Z 362.856,A -85,B 0,C 180,E1 -5927.455,E2 -5927.455} C_VEL
LIN {X 0,Y 503.698,Z 372.247,A -85,B 0,C 180,E1 -5928.327,E2 -5928.327} C_VEL
LIN {X 0,Y 503.438,Z 381.125,A -85,B 0,C 180,E1 -5929.34,E2 -5929.34} C_VEL
LIN {X 0,Y 503.131,Z 389.751,A -85,B 0,C 180,E1 -5930.553,E2 -5930.553} C_VEL
LIN {X 0,Y 502.885,Z 396.63,A -85,B 0,C 180,E1 -5931.764,E2 -5931.764} C_VEL
LIN {X 0,Y 502.671,Z 402.441,A -85,B 0,C 180,E1 -5933.063,E2 -5933.063} C_VEL
LIN {X 0,Y 502.576,Z 406.94,A -85,B 0,C 180,E1 -5934.382,E2 -5934.382} C_VEL
LIN {X 0,Y 502.459,Z 409.087,A -85,B 0,C 180,E1 -5935.186,E2 -5935.186} C_VEL
LIN {X 0,Y 502.445,Z 410.778,A -85,B 0,C 180,E1 -5935.989,E2 -5935.989} C_VEL
LIN {X 0,Y 502.322,Z 412.909,A -85,B 0,C 180,E1 -5937.594,E2 -5937.594} C_VEL
LIN {X 0,Y 502.329,Z 413.396,A -85,B 0,C 180,E1 -5938.396,E2 -5938.396} C_VEL
LIN {X 0,Y 502.273,Z 413.162,A -85,B 0,C 180,E1 -5940,E2 -5940} C_VEL
LIN {X 0,Y 502.336,Z 411.365,A -85,B 0,C 180,E1 -5941.603,E2 -5941.603} C_VEL
LIN {X 0,Y 502.333,Z 409.866,A -85,B 0,C 180,E1 -5942.405,E2 -5942.405} C_VEL
LIN {X 0,Y 502.565,Z 406.787,A -85,B 0,C 180,E1 -5943.608,E2 -5943.608} C_VEL
LIN {X 0,Y 502.56,Z 402.705,A -85,B 0,C 180,E1 -5944.813,E2 -5944.813} C_VEL
LIN {X 0,Y 502.798,Z 396.422,A -85,B 0,C 180,E1 -5946.219,E2 -5946.219} C_VEL
LIN {X 0,Y 502.999,Z 389.598,A -85,B 0,C 180,E1 -5947.426,E2 -5947.426} C_VEL
LIN {X 0,Y 503.204,Z 381.081,A -85,B 0,C 180,E1 -5948.635,E2 -5948.635} C_VEL
LIN {X 0,Y 503.557,Z 372.301,A -85,B 0,C 180,E1 -5949.641,E2 -5949.641} C_VEL
LIN {X 0,Y 503.878,Z 362.692,A -85,B 0,C 180,E1 -5950.548,E2 -5950.548} C_VEL
LIN {X 0,Y 504.115,Z 352.227,A -85,B 0,C 180,E1 -5951.353,E2 -5951.353} C_VEL
LIN {X 0,Y 504.412,Z 340.473,A -85,B 0,C 180,E1 -5952.063,E2 -5952.063} C_VEL
LIN {X 0,Y 503.987,Z 337.03,A -85,B 0,C 180,E1 -5952.256,E2 -5952.256} C_VEL
LIN {X 0,Y 502.859,Z 332.848,A -85,B 0,C 180,E1 -5952.511,E2 -5952.511} C_VEL
LIN {X 0,Y 502.853,Z 332.85,A -85,B 0,C 180,E1 -5955.399,E2 -5955.399} C_VEL
LIN {X 0,Y 502.827,Z 332.85,A -85,B 0,C 180,E1 -5958.752,E2 -5958.752} C_VEL
LIN {X 0,Y 502.787,Z 332.855,A -85,B 0,C 180,E1 -5961.311,E2 -5961.311} C_VEL
LIN {X 0,Y 502.789,Z 332.855,A -85,B 0,C 180,E1 -5963.914,E2 -5963.914} C_VEL
LIN {X 0,Y 502.868,Z 332.846,A -85,B 0,C 180,E1 -5966.566,E2 -5966.566} C_VEL
LIN {X 0,Y 502.828,Z 332.851,A -85,B 0,C 180,E1 -5969.287,E2 -5969.287} C_VEL
LIN {X 0,Y 502.79,Z 332.854,A -85,B 0,C 180,E1 -5972.084,E2 -5972.084} C_VEL
LIN {X 0,Y 502.804,Z 332.857,A -85,B 0,C 180,E1 -5974.965,E2 -5974.965} C_VEL
LIN {X 0,Y 502.797,Z 332.852,A -85,B 0,C 180,E1 -5977.954,E2 -5977.954} C_VEL
LIN {X 0,Y 502.83,Z 332.849,A -85,B 0,C 180,E1 -5981.065,E2 -5981.065} C_VEL
LIN {X 0,Y 502.803,Z 332.853,A -85,B 0,C 180,E1 -5984.532,E2 -5984.532} C_VEL
LIN {X 0,Y 502.832,Z 332.85,A -85,B 0,C 180,E1 -5987.864,E2 -5987.864} C_VEL
LIN {X 0,Y 502.796,Z 332.854,A -85,B 0,C 180,E1 -5991.232,E2 -5991.232} C_VEL
LIN {X 0,Y 502.776,Z 332.856,A -85,B 0,C 180,E1 -5994.169,E2 -5994.169} C_VEL
LIN {X 0,Y 502.778,Z 332.854,A -85,B 0,C 180,E1 -5994.713,E2 -5994.713} C_VEL
LIN {X 0,Y 502.134,Z 332.936,A -85,B 0,C 180,E1 -5995.382,E2 -5995.382} C_VEL
LIN {X 0,Y 499.272,Z 333.296,A -85,B 0,C 180,E1 -5996.468,E2 -5996.468} C_VEL
LIN {X 0,Y 496.85,Z 333.594,A -85,B 0,C 180,E1 -5997.344,E2 -5997.344} C_VEL
LIN {X 0,Y 495.829,Z 333.725,A -85,B 0,C 180,E1 -5998.02,E2 -5998.02} C_VEL
LIN {X 0,Y 495.757,Z 333.733,A -85,B 0,C 180,E1 -5998.249,E2 -5998.249} C_VEL
LIN {X 0,Y 495.789,Z 333.729,A -85,B 0,C 180,E1 -6001.507,E2 -6001.507} C_VEL
LIN {X 0,Y 495.793,Z 333.726,A -85,B 0,C 180,E1 -6003.932,E2 -6003.932} C_VEL
LIN {X 0,Y 495.76,Z 333.732,A -85,B 0,C 180,E1 -6007.139,E2 -6007.139} C_VEL
LIN {X 0,Y 495.779,Z 333.729,A -85,B 0,C 180,E1 -6010.11,E2 -6010.11} C_VEL
LIN {X 0,Y 495.788,Z 333.726,A -85,B 0,C 180,E1 -6012.681,E2 -6012.681} C_VEL
LIN {X 0,Y 495.792,Z 333.726,A -85,B 0,C 180,E1 -6015.217,E2 -6015.217} C_VEL
LIN {X 0,Y 495.854,Z 333.718,A -85,B 0,C 180,E1 -6018.555,E2 -6018.555} C_VEL
LIN {X 0,Y 495.874,Z 333.715,A -85,B 0,C 180,E1 -6021.852,E2 -6021.852} C_VEL
LIN {X 0,Y 495.892,Z 333.716,A -85,B 0,C 180,E1 -6024.307,E2 -6024.307} C_VEL
LIN {X 0,Y 495.995,Z 333.7,A -85,B 0,C 180,E1 -6027.564,E2 -6027.564} C_VEL
LIN {X 0,Y 496.006,Z 333.697,A -85,B 0,C 180,E1 -6030.812,E2 -6030.812} C_VEL
LIN {X 0,Y 495.846,Z 333.721,A -85,B 0,C 180,E1 -6033.25,E2 -6033.25} C_VEL
LIN {X 0,Y 495.863,Z 333.718,A -85,B 0,C 180,E1 -6036.511,E2 -6036.511} C_VEL
LIN {X 0,Y 495.845,Z 333.722,A -85,B 0,C 180,E1 -6038.97,E2 -6038.97} C_VEL
LIN {X 0,Y 495.83,Z 333.724,A -85,B 0,C 180,E1 -6042.035,E2 -6042.035} C_VEL
LIN {X 0,Y 495.825,Z 333.722,A -85,B 0,C 180,E1 -6045.452,E2 -6045.452} C_VEL
LIN {X 0,Y 495.808,Z 333.723,A -85,B 0,C 180,E1 -6048.247,E2 -6048.247} C_VEL
LIN {X 0,Y 495.776,Z 333.729,A -85,B 0,C 180,E1 -6050.757,E2 -6050.757} C_VEL
LIN {X 0,Y 495.75,Z 333.732,A -85,B 0,C 180,E1 -6053.387,E2 -6053.387} C_VEL
LIN {X 0,Y 495.793,Z 333.728,A -85,B 0,C 180,E1 -6056.068,E2 -6056.068} C_VEL
LIN {X 0,Y 495.774,Z 333.728,A -85,B 0,C 180,E1 -6058.815,E2 -6058.815} C_VEL
LIN {X 0,Y 495.759,Z 333.734,A -85,B 0,C 180,E1 -6061.726,E2 -6061.726} C_VEL
LIN {X 0,Y 495.771,Z 333.727,A -85,B 0,C 180,E1 -6064.694,E2 -6064.694} C_VEL
LIN {X 0,Y 495.731,Z 333.734,A -85,B 0,C 180,E1 -6067.562,E2 -6067.562} C_VEL
LIN {X 0,Y 495.769,Z 333.732,A -85,B 0,C 180,E1 -6070.7,E2 -6070.7} C_VEL
LIN {X 0,Y 495.738,Z 333.734,A -85,B 0,C 180,E1 -6073.696,E2 -6073.696} C_VEL
LIN {X 0,Y 495.732,Z 333.735,A -85,B 0,C 180,E1 -6076.306,E2 -6076.306} C_VEL
LIN {X 0,Y 495.77,Z 333.733,A -85,B 0,C 180,E1 -6079.3,E2 -6079.3} C_VEL
LIN {X 0,Y 495.733,Z 333.732,A -85,B 0,C 180,E1 -6082.439,E2 -6082.439} C_VEL
LIN {X 0,Y 495.785,Z 333.726,A -85,B 0,C 180,E1 -6085.457,E2 -6085.457} C_VEL
LIN {X 0,Y 495.76,Z 333.733,A -85,B 0,C 180,E1 -6088.364,E2 -6088.364} C_VEL
LIN {X 0,Y 495.792,Z 333.729,A -85,B 0,C 180,E1 -6091.507,E2 -6091.507} C_VEL
LIN {X 0,Y 495.796,Z 333.727,A -85,B 0,C 180,E1 -6093.933,E2 -6093.933} C_VEL
LIN {X 0,Y 495.765,Z 333.734,A -85,B 0,C 180,E1 -6097.14,E2 -6097.14} C_VEL
LIN {X 0,Y 495.774,Z 333.727,A -85,B 0,C 180,E1 -6100.11,E2 -6100.11} C_VEL
LIN {X 0,Y 495.785,Z 333.73,A -85,B 0,C 180,E1 -6102.681,E2 -6102.681} C_VEL
LIN {X 0,Y 495.796,Z 333.725,A -85,B 0,C 180,E1 -6105.217,E2 -6105.217} C_VEL
LIN {X 0,Y 495.857,Z 333.718,A -85,B 0,C 180,E1 -6108.555,E2 -6108.555} C_VEL
LIN {X 0,Y 495.879,Z 333.715,A -85,B 0,C 180,E1 -6111.852,E2 -6111.852} C_VEL
LIN {X 0,Y 495.901,Z 333.712,A -85,B 0,C 180,E1 -6114.307,E2 -6114.307} C_VEL
LIN {X 0,Y 495.997,Z 333.698,A -85,B 0,C 180,E1 -6117.564,E2 -6117.564} C_VEL
LIN {X 0,Y 496.011,Z 333.698,A -85,B 0,C 180,E1 -6120.812,E2 -6120.812} C_VEL
LIN {X 0,Y 495.847,Z 333.72,A -85,B 0,C 180,E1 -6123.25,E2 -6123.25} C_VEL
LIN {X 0,Y 495.866,Z 333.717,A -85,B 0,C 180,E1 -6126.511,E2 -6126.511} C_VEL
LIN {X 0,Y 495.841,Z 333.723,A -85,B 0,C 180,E1 -6128.97,E2 -6128.97} C_VEL
LIN {X 0,Y 495.834,Z 333.721,A -85,B 0,C 180,E1 -6132.035,E2 -6132.035} C_VEL
LIN {X 0,Y 495.83,Z 333.719,A -85,B 0,C 180,E1 -6135.452,E2 -6135.452} C_VEL
LIN {X 0,Y 495.813,Z 333.725,A -85,B 0,C 180,E1 -6138.247,E2 -6138.247} C_VEL
LIN {X 0,Y 495.78,Z 333.727,A -85,B 0,C 180,E1 -6140.756,E2 -6140.756} C_VEL
LIN {X 0,Y 495.753,Z 333.734,A -85,B 0,C 180,E1 -6143.387,E2 -6143.387} C_VEL
LIN {X 0,Y 495.796,Z 333.726,A -85,B 0,C 180,E1 -6146.068,E2 -6146.068} C_VEL
LIN {X 0,Y 495.777,Z 333.729,A -85,B 0,C 180,E1 -6148.815,E2 -6148.815} C_VEL
LIN {X 0,Y 495.76,Z 333.731,A -85,B 0,C 180,E1 -6151.725,E2 -6151.725} C_VEL
LIN {X 0,Y 495.78,Z 333.726,A -85,B 0,C 180,E1 -6154.695,E2 -6154.695} C_VEL
LIN {X 0,Y 495.736,Z 333.736,A -85,B 0,C 180,E1 -6157.561,E2 -6157.561} C_VEL
LIN {X 0,Y 495.771,Z 333.731,A -85,B 0,C 180,E1 -6160.7,E2 -6160.7} C_VEL
LIN {X 0,Y 495.739,Z 333.734,A -85,B 0,C 180,E1 -6164.001,E2 -6164.001} C_VEL
LIN {X 0,Y 495.738,Z 333.733,A -85,B 0,C 180,E1 -6167.118,E2 -6167.118} C_VEL
LIN {X 0,Y 495.766,Z 333.823,A -85,B 0,C 180,E1 -6170.158,E2 -6170.158} C_VEL
LIN {X 0,Y 498.002,Z 344.853,A -85,B 0,C 180,E1 -6173.12,E2 -6173.12} C_VEL
LIN {X 0,Y 498.319,Z 349.031,A -85,B 0,C 180,E1 -6174.176,E2 -6174.176} C_VEL
LIN {X 0,Y 497.696,Z 362.099,A -85,B 0,C 180,E1 -6177.307,E2 -6177.307} C_VEL
LIN {X 0,Y 497.181,Z 375.155,A -85,B 0,C 180,E1 -6180.346,E2 -6180.346} C_VEL
LIN {X 0,Y 496.81,Z 389.221,A -85,B 0,C 180,E1 -6183.538,E2 -6183.538} C_VEL
LIN {X 0,Y 496.393,Z 403.276,A -85,B 0,C 180,E1 -6186.645,E2 -6186.645} C_VEL
LIN {X 0,Y 496.06,Z 417.397,A -85,B 0,C 180,E1 -6189.689,E2 -6189.689} C_VEL
LIN {X 0,Y 495.847,Z 431.666,A -85,B 0,C 180,E1 -6192.683,E2 -6192.683} C_VEL
LIN {X 0,Y 495.577,Z 444.815,A -85,B 0,C 180,E1 -6195.473,E2 -6195.473} C_VEL
LIN {X 0,Y 497.046,Z 458.644,A -85,B 0,C 180,E1 -6195.843,E2 -6195.843} C_VEL
LIN {X 0,Y 497.516,Z 463.229,A -85,B 0,C 180,E1 -6196,E2 -6196} C_VEL
LIN {X 0,Y 497.144,Z 475.903,A -85,B 0,C 180,E1 -6196.511,E2 -6196.511} C_VEL
LIN {X 0,Y 496.775,Z 487.676,A -85,B 0,C 180,E1 -6197.146,E2 -6197.146} C_VEL
LIN {X 0,Y 496.458,Z 499.203,A -85,B 0,C 180,E1 -6197.948,E2 -6197.948} C_VEL
LIN {X 0,Y 496.033,Z 509.853,A -85,B 0,C 180,E1 -6198.869,E2 -6198.869} C_VEL
LIN {X 0,Y 495.76,Z 518.604,A -85,B 0,C 180,E1 -6199.793,E2 -6199.793} C_VEL
LIN {X 0,Y 495.529,Z 526.69,A -85,B 0,C 180,E1 -6200.819,E2 -6200.819} C_VEL
LIN {X 0,Y 495.376,Z 534.627,A -85,B 0,C 180,E1 -6202.049,E2 -6202.049} C_VEL
LIN {X 0,Y 495.213,Z 541.906,A -85,B 0,C 180,E1 -6203.481,E2 -6203.481} C_VEL
LIN {X 0,Y 495.176,Z 546.764,A -85,B 0,C 180,E1 -6204.707,E2 -6204.707} C_VEL
LIN {X 0,Y 495.217,Z 550.482,A -85,B 0,C 180,E1 -6205.931,E2 -6205.931} C_VEL
LIN {X 0,Y 495.145,Z 552.378,A -85,B 0,C 180,E1 -6206.745,E2 -6206.745} C_VEL
LIN {X 0,Y 495.129,Z 553.81,A -85,B 0,C 180,E1 -6207.559,E2 -6207.559} C_VEL
LIN {X 0,Y 495.083,Z 554.817,A -85,B 0,C 180,E1 -6208.373,E2 -6208.373} C_VEL
LIN {X 0,Y 495.125,Z 555.619,A -85,B 0,C 180,E1 -6210,E2 -6210} C_VEL
LIN {X 0,Y 495.136,Z 555.375,A -85,B 0,C 180,E1 -6210.813,E2 -6210.813} C_VEL
LIN {X 0,Y 495.096,Z 554.716,A -85,B 0,C 180,E1 -6211.627,E2 -6211.627} C_VEL
LIN {X 0,Y 495.147,Z 553.651,A -85,B 0,C 180,E1 -6212.44,E2 -6212.44} C_VEL
LIN {X 0,Y 495.169,Z 552.16,A -85,B 0,C 180,E1 -6213.255,E2 -6213.255} C_VEL
LIN {X 0,Y 495.202,Z 549.056,A -85,B 0,C 180,E1 -6214.477,E2 -6214.477} C_VEL
LIN {X 0,Y 495.25,Z 544.863,A -85,B 0,C 180,E1 -6215.701,E2 -6215.701} C_VEL
LIN {X 0,Y 495.317,Z 538.533,A -85,B 0,C 180,E1 -6217.111,E2 -6217.111} C_VEL
LIN {X 0,Y 495.455,Z 531.402,A -85,B 0,C 180,E1 -6218.36,E2 -6218.36} C_VEL
LIN {X 0,Y 495.634,Z 522.687,A -85,B 0,C 180,E1 -6219.591,E2 -6219.591} C_VEL
LIN {X 0,Y 495.902,Z 512.742,A -85,B 0,C 180,E1 -6220.72,E2 -6220.72} C_VEL
LIN {X 0,Y 496.326,Z 501.574,A -85,B 0,C 180,E1 -6221.745,E2 -6221.745} C_VEL
LIN {X 0,Y 496.581,Z 490.875,A -85,B 0,C 180,E1 -6222.537,E2 -6222.537} C_VEL
LIN {X 0,Y 496.946,Z 477.981,A -85,B 0,C 180,E1 -6223.286,E2 -6223.286} C_VEL
LIN {X 0,Y 497.336,Z 465.191,A -85,B 0,C 180,E1 -6223.848,E2 -6223.848} C_VEL
LIN {X 0,Y 497.204,Z 460.323,A -85,B 0,C 180,E1 -6224.021,E2 -6224.021} C_VEL
LIN {X 0,Y 496.103,Z 450.33,A -85,B 0,C 180,E1 -6224.328,E2 -6224.328} C_VEL
LIN {X 0,Y 495.566,Z 442.391,A -85,B 0,C 180,E1 -6224.527,E2 -6224.527} C_VEL
LIN {X 0,Y 495.758,Z 426.262,A -85,B 0,C 180,E1 -6227.746,E2 -6227.746} C_VEL
LIN {X 0,Y 495.906,Z 410.209,A -85,B 0,C 180,E1 -6230.968,E2 -6230.968} C_VEL
LIN {X 0,Y 496.044,Z 395.154,A -85,B 0,C 180,E1 -6234.038,E2 -6234.038} C_VEL
LIN {X 0,Y 496.21,Z 380.124,A -85,B 0,C 180,E1 -6237.179,E2 -6237.179} C_VEL
LIN {X 0,Y 496.371,Z 365.921,A -85,B 0,C 180,E1 -6240.267,E2 -6240.267} C_VEL
LIN {X 0,Y 496.597,Z 354.126,A -85,B 0,C 180,E1 -6242.965,E2 -6242.965} C_VEL
LIN {X 0,Y 497.223,Z 342.321,A -85,B 0,C 180,E1 -6245.851,E2 -6245.851} C_VEL
LIN {X 0,Y 496.265,Z 336.355,A -85,B 0,C 180,E1 -6247.527,E2 -6247.527} C_VEL
LIN {X 0,Y 495.783,Z 333.733,A -85,B 0,C 180,E1 -6248.329,E2 -6248.329} C_VEL
LIN {X 0,Y 495.76,Z 333.734,A -85,B 0,C 180,E1 -6251.293,E2 -6251.293} C_VEL
LIN {X 0,Y 495.738,Z 333.736,A -85,B 0,C 180,E1 -6254.001,E2 -6254.001} C_VEL
LIN {X 0,Y 495.73,Z 333.737,A -85,B 0,C 180,E1 -6257.117,E2 -6257.117} C_VEL
LIN {X 0,Y 495.762,Z 333.733,A -85,B 0,C 180,E1 -6259.953,E2 -6259.953} C_VEL
LIN {X 0,Y 495.734,Z 333.734,A -85,B 0,C 180,E1 -6262.553,E2 -6262.553} C_VEL
LIN {X 0,Y 495.788,Z 333.729,A -85,B 0,C 180,E1 -6265.457,E2 -6265.457} C_VEL
LIN {X 0,Y 495.76,Z 333.734,A -85,B 0,C 180,E1 -6268.364,E2 -6268.364} C_VEL
LIN {X 0,Y 495.792,Z 333.728,A -85,B 0,C 180,E1 -6271.507,E2 -6271.507} C_VEL
LIN {X 0,Y 495.785,Z 333.729,A -85,B 0,C 180,E1 -6273.932,E2 -6273.932} C_VEL
LIN {X 0,Y 495.764,Z 333.734,A -85,B 0,C 180,E1 -6277.14,E2 -6277.14} C_VEL
LIN {X 0,Y 495.776,Z 333.732,A -85,B 0,C 180,E1 -6280.11,E2 -6280.11} C_VEL
LIN {X 0,Y 495.786,Z 333.732,A -85,B 0,C 180,E1 -6282.681,E2 -6282.681} C_VEL
LIN {X 0,Y 495.826,Z 333.915,A -85,B 0,C 180,E1 -6285.349,E2 -6285.349} C_VEL
LIN {X 0,Y 497.739,Z 341.789,A -85,B 0,C 180,E1 -6285.798,E2 -6285.798} C_VEL
LIN {X 0,Y 497.419,Z 353.725,A -85,B 0,C 180,E1 -6286.519,E2 -6286.519} C_VEL
LIN {X 0,Y 497.12,Z 363.797,A -85,B 0,C 180,E1 -6287.288,E2 -6287.288} C_VEL
LIN {X 0,Y 496.807,Z 373.118,A -85,B 0,C 180,E1 -6288.163,E2 -6288.163} C_VEL
LIN {X 0,Y 496.53,Z 382.017,A -85,B 0,C 180,E1 -6289.19,E2 -6289.19} C_VEL
LIN {X 0,Y 496.195,Z 390.666,A -85,B 0,C 180,E1 -6290.42,E2 -6290.42} C_VEL
LIN {X 0,Y 495.931,Z 397.589,A -85,B 0,C 180,E1 -6291.648,E2 -6291.648} C_VEL
LIN {X 0,Y 495.696,Z 403.415,A -85,B 0,C 180,E1 -6292.965,E2 -6292.965} C_VEL
LIN {X 0,Y 495.59,Z 407.931,A -85,B 0,C 180,E1 -6294.303,E2 -6294.303} C_VEL
LIN {X 0,Y 495.456,Z 410.091,A -85,B 0,C 180,E1 -6295.118,E2 -6295.118} C_VEL
LIN {X 0,Y 495.43,Z 411.787,A -85,B 0,C 180,E1 -6295.933,E2 -6295.933} C_VEL
LIN {X 0,Y 495.3,Z 413.921,A -85,B 0,C 180,E1 -6297.56,E2 -6297.56} C_VEL
LIN {X 0,Y 495.315,Z 414.407,A -85,B 0,C 180,E1 -6298.374,E2 -6298.374} C_VEL
LIN {X 0,Y 495.264,Z 414.489,A -85,B 0,C 180,E1 -6299.187,E2 -6299.187} C_VEL
LIN {X 0,Y 495.268,Z 413.459,A -85,B 0,C 180,E1 -6300.813,E2 -6300.813} C_VEL
LIN {X 0,Y 495.322,Z 412.364,A -85,B 0,C 180,E1 -6301.626,E2 -6301.626} C_VEL
LIN {X 0,Y 495.31,Z 410.856,A -85,B 0,C 180,E1 -6302.44,E2 -6302.44} C_VEL
LIN {X 0,Y 495.557,Z 407.764,A -85,B 0,C 180,E1 -6303.659,E2 -6303.659} C_VEL
LIN {X 0,Y 495.551,Z 403.668,A -85,B 0,C 180,E1 -6304.881,E2 -6304.881} C_VEL
LIN {X 0,Y 495.81,Z 397.368,A -85,B 0,C 180,E1 -6306.307,E2 -6306.307} C_VEL
LIN {X 0,Y 496.031,Z 390.531,A -85,B 0,C 180,E1 -6307.531,E2 -6307.531} C_VEL
LIN {X 0,Y 496.257,Z 381.993,A -85,B 0,C 180,E1 -6308.757,E2 -6308.757} C_VEL
LIN {X 0,Y 496.627,Z 373.203,A -85,B 0,C 180,E1 -6309.777,E2 -6309.777} C_VEL
LIN {X 0,Y 497.004,Z 362.409,A -85,B 0,C 180,E1 -6310.799,E2 -6310.799} C_VEL
LIN {X 0,Y 497.273,Z 351.785,A -85,B 0,C 180,E1 -6311.602,E2 -6311.602} C_VEL
LIN {X 0,Y 497.553,Z 340.299,A -85,B 0,C 180,E1 -6312.289,E2 -6312.289} C_VEL
LIN {X 0,Y 495.82,Z 333.724,A -85,B 0,C 180,E1 -6312.686,E2 -6312.686} C_VEL
LIN {X 0,Y 495.811,Z 333.727,A -85,B 0,C 180,E1 -6315.624,E2 -6315.624} C_VEL
LIN {X 0,Y 495.783,Z 333.731,A -85,B 0,C 180,E1 -6319.028,E2 -6319.028} C_VEL
LIN {X 0,Y 495.747,Z 333.731,A -85,B 0,C 180,E1 -6321.629,E2 -6321.629} C_VEL
LIN {X 0,Y 495.782,Z 333.728,A -85,B 0,C 180,E1 -6324.873,E2 -6324.873} C_VEL
LIN {X 0,Y 495.818,Z 333.723,A -85,B 0,C 180,E1 -6326.974,E2 -6326.974} C_VEL
LIN {X 0,Y 495.769,Z 333.73,A -85,B 0,C 180,E1 -6330.147,E2 -6330.147} C_VEL
LIN {X 0,Y 495.796,Z 333.729,A -85,B 0,C 180,E1 -6333.244,E2 -6333.244} C_VEL
LIN {X 0,Y 495.723,Z 333.732,A -85,B 0,C 180,E1 -6336.088,E2 -6336.088} C_VEL
LIN {X 0,Y 495.772,Z 333.732,A -85,B 0,C 180,E1 -6338.769,E2 -6338.769} C_VEL
LIN {X 0,Y 495.764,Z 333.732,A -85,B 0,C 180,E1 -6341.78,E2 -6341.78} C_VEL
LIN {X 0,Y 495.752,Z 333.732,A -85,B 0,C 180,E1 -6345.139,E2 -6345.139} C_VEL
LIN {X 0,Y 495.78,Z 333.727,A -85,B 0,C 180,E1 -6348.221,E2 -6348.221} C_VEL
LIN {X 0,Y 495.752,Z 333.731,A -85,B 0,C 180,E1 -6351.408,E2 -6351.408} C_VEL
LIN {X 0,Y 495.745,Z 333.733,A -85,B 0,C 180,E1 -6354.713,E2 -6354.713} C_VEL
LIN {X 0,Y 495.77,Z 333.728,A -85,B 0,C 180,E1 -6357.406,E2 -6357.406} C_VEL
LIN {X 0,Y 495.757,Z 333.733,A -85,B 0,C 180,E1 -6358.249,E2 -6358.249} C_VEL
LIN {X 0,Y 495.124,Z 333.818,A -85,B 0,C 180,E1 -6358.927,E2 -6358.927} C_VEL
LIN {X 0,Y 492.296,Z 334.174,A -85,B 0,C 180,E1 -6360.028,E2 -6360.028} C_VEL
LIN {X 0,Y 489.878,Z 334.471,A -85,B 0,C 180,E1 -6360.915,E2 -6360.915} C_VEL
LIN {X 0,Y 488.828,Z 334.597,A -85,B 0,C 180,E1 -6361.6,E2 -6361.6} C_VEL
LIN {X 0,Y 488.737,Z 334.606,A -85,B 0,C 180,E1 -6361.832,E2 -6361.832} C_VEL
LIN {X 0,Y 488.749,Z 334.603,A -85,B 0,C 180,E1 -6364.444,E2 -6364.444} C_VEL
LIN {X 0,Y 488.723,Z 334.608,A -85,B 0,C 180,E1 -6367.153,E2 -6367.153} C_VEL
LIN {X 0,Y 488.73,Z 334.605,A -85,B 0,C 180,E1 -6369.811,E2 -6369.811} C_VEL
LIN {X 0,Y 488.736,Z 334.607,A -85,B 0,C 180,E1 -6372.423,E2 -6372.423} C_VEL
LIN {X 0,Y 488.764,Z 334.601,A -85,B 0,C 180,E1 -6375,E2 -6375} C_VEL
LIN {X 0,Y 488.807,Z 334.596,A -85,B 0,C 180,E1 -6378.388,E2 -6378.388} C_VEL
LIN {X 0,Y 488.819,Z 334.595,A -85,B 0,C 180,E1 -6381.734,E2 -6381.734} C_VEL
LIN {X 0,Y 488.851,Z 334.593,A -85,B 0,C 180,E1 -6384.224,E2 -6384.224} C_VEL
LIN {X 0,Y 488.963,Z 334.576,A -85,B 0,C 180,E1 -6387.529,E2 -6387.529} C_VEL
LIN {X 0,Y 488.956,Z 334.576,A -85,B 0,C 180,E1 -6390.824,E2 -6390.824} C_VEL
LIN {X 0,Y 488.964,Z 334.576,A -85,B 0,C 180,E1 -6392.471,E2 -6392.471} C_VEL
LIN {X 0,Y 488.85,Z 334.591,A -85,B 0,C 180,E1 -6395.776,E2 -6395.776} C_VEL
LIN {X 0,Y 488.82,Z 334.596,A -85,B 0,C 180,E1 -6398.266,E2 -6398.266} C_VEL
LIN {X 0,Y 488.808,Z 334.596,A -85,B 0,C 180,E1 -6401.613,E2 -6401.613} C_VEL
LIN {X 0,Y 488.764,Z 334.6,A -85,B 0,C 180,E1 -6405,E2 -6405} C_VEL
LIN {X 0,Y 488.757,Z 334.601,A -85,B 0,C 180,E1 -6408.442,E2 -6408.442} C_VEL
LIN {X 0,Y 488.708,Z 334.611,A -85,B 0,C 180,E1 -6411.071,E2 -6411.071} C_VEL
LIN {X 0,Y 488.691,Z 334.61,A -85,B 0,C 180,E1 -6413.746,E2 -6413.746} C_VEL
LIN {X 0,Y 488.794,Z 334.599,A -85,B 0,C 180,E1 -6416.944,E2 -6416.944} C_VEL
LIN {X 0,Y 488.712,Z 334.609,A -85,B 0,C 180,E1 -6420.363,E2 -6420.363} C_VEL
LIN {X 0,Y 488.737,Z 334.61,A -85,B 0,C 180,E1 -6423.484,E2 -6423.484} C_VEL
LIN {X 0,Y 488.684,Z 334.61,A -85,B 0,C 180,E1 -6426.355,E2 -6426.355} C_VEL
LIN {X 0,Y 488.703,Z 334.61,A -85,B 0,C 180,E1 -6429.255,E2 -6429.255} C_VEL
LIN {X 0,Y 488.738,Z 334.608,A -85,B 0,C 180,E1 -6432.521,E2 -6432.521} C_VEL
LIN {X 0,Y 488.715,Z 334.607,A -85,B 0,C 180,E1 -6435.199,E2 -6435.199} C_VEL
LIN {X 0,Y 488.711,Z 334.607,A -85,B 0,C 180,E1 -6438.4,E2 -6438.4} C_VEL
LIN {X 0,Y 488.707,Z 334.61,A -85,B 0,C 180,E1 -6440.948,E2 -6440.948} C_VEL
LIN {X 0,Y 488.682,Z 334.61,A -85,B 0,C 180,E1 -6443.868,E2 -6443.868} C_VEL
LIN {X 0,Y 488.742,Z 334.606,A -85,B 0,C 180,E1 -6446.878,E2 -6446.878} C_VEL
LIN {X 0,Y 488.728,Z 334.609,A -85,B 0,C 180,E1 -6449.781,E2 -6449.781} C_VEL
LIN {X 0,Y 488.797,Z 334.598,A -85,B 0,C 180,E1 -6453.057,E2 -6453.057} C_VEL
LIN {X 0,Y 488.693,Z 334.609,A -85,B 0,C 180,E1 -6456.255,E2 -6456.255} C_VEL
LIN {X 0,Y 488.751,Z 334.604,A -85,B 0,C 180,E1 -6459.176,E2 -6459.176} C_VEL
LIN {X 0,Y 488.733,Z 334.608,A -85,B 0,C 180,E1 -6462.423,E2 -6462.423} C_VEL
LIN {X 0,Y 488.768,Z 334.601,A -85,B 0,C 180,E1 -6465,E2 -6465} C_VEL
LIN {X 0,Y 488.811,Z 334.596,A -85,B 0,C 180,E1 -6468.388,E2 -6468.388} C_VEL
LIN {X 0,Y 488.824,Z 334.595,A -85,B 0,C 180,E1 -6471.734,E2 -6471.734} C_VEL
LIN {X 0,Y 488.86,Z 334.589,A -85,B 0,C 180,E1 -6474.224,E2 -6474.224} C_VEL
LIN {X 0,Y 488.965,Z 334.574,A -85,B 0,C 180,E1 -6477.529,E2 -6477.529} C_VEL
LIN {X 0,Y 488.96,Z 334.576,A -85,B 0,C 180,E1 -6480.824,E2 -6480.824} C_VEL
LIN {X 0,Y 488.967,Z 334.577,A -85,B 0,C 180,E1 -6482.471,E2 -6482.471} C_VEL
LIN {X 0,Y 488.852,Z 334.593,A -85,B 0,C 180,E1 -6485.776,E2 -6485.776} C_VEL
LIN {X 0,Y 488.791,Z 334.598,A -85,B 0,C 180,E1 -6488.267,E2 -6488.267} C_VEL
LIN {X 0,Y 488.812,Z 334.594,A -85,B 0,C 180,E1 -6491.612,E2 -6491.612} C_VEL
LIN {X 0,Y 488.768,Z 334.599,A -85,B 0,C 180,E1 -6495,E2 -6495} C_VEL
LIN {X 0,Y 488.761,Z 334.602,A -85,B 0,C 180,E1 -6498.442,E2 -6498.442} C_VEL
LIN {X 0,Y 488.713,Z 334.61,A -85,B 0,C 180,E1 -6501.071,E2 -6501.071} C_VEL
LIN {X 0,Y 488.694,Z 334.611,A -85,B 0,C 180,E1 -6503.746,E2 -6503.746} C_VEL
LIN {X 0,Y 488.797,Z 334.599,A -85,B 0,C 180,E1 -6506.944,E2 -6506.944} C_VEL
LIN {X 0,Y 488.715,Z 334.61,A -85,B 0,C 180,E1 -6510.363,E2 -6510.363} C_VEL
LIN {X 0,Y 488.741,Z 334.605,A -85,B 0,C 180,E1 -6513.484,E2 -6513.484} C_VEL
LIN {X 0,Y 488.692,Z 334.609,A -85,B 0,C 180,E1 -6516.355,E2 -6516.355} C_VEL
LIN {X 0,Y 488.706,Z 334.612,A -85,B 0,C 180,E1 -6519.254,E2 -6519.254} C_VEL
LIN {X 0,Y 488.711,Z 334.608,A -85,B 0,C 180,E1 -6521.6,E2 -6521.6} C_VEL
LIN {X 0,Y 488.717,Z 334.609,A -85,B 0,C 180,E1 -6524.801,E2 -6524.801} C_VEL
LIN {X 0,Y 488.699,Z 334.611,A -85,B 0,C 180,E1 -6527.475,E2 -6527.475} C_VEL
LIN {X 0,Y 488.729,Z 334.717,A -85,B 0,C 180,E1 -6529.878,E2 -6529.878} C_VEL
LIN {X 0,Y 490.698,Z 344.442,A -85,B 0,C 180,E1 -6532.543,E2 -6532.543} C_VEL
LIN {X 0,Y 491.413,Z 348.768,A -85,B 0,C 180,E1 -6533.684,E2 -6533.684} C_VEL
LIN {X 0,Y 490.851,Z 360.606,A -85,B 0,C 180,E1 -6536.578,E2 -6536.578} C_VEL
LIN {X 0,Y 490.331,Z 373.287,A -85,B 0,C 180,E1 -6539.595,E2 -6539.595} C_VEL
LIN {X 0,Y 489.89,Z 387.136,A -85,B 0,C 180,E1 -6542.806,E2 -6542.806} C_VEL
LIN {X 0,Y 489.393,Z 402.597,A -85,B 0,C 180,E1 -6546.29,E2 -6546.29} C_VEL
LIN {X 0,Y 489.017,Z 417.002,A -85,B 0,C 180,E1 -6549.452,E2 -6549.452} C_VEL
LIN {X 0,Y 488.759,Z 430.781,A -85,B 0,C 180,E1 -6552.424,E2 -6552.424} C_VEL
LIN {X 0,Y 488.478,Z 443.943,A -85,B 0,C 180,E1 -6555.257,E2 -6555.257} C_VEL
LIN {X 0,Y 490.075,Z 459.245,A -85,B 0,C 180,E1 -6555.691,E2 -6555.691} C_VEL
LIN {X 0,Y 490.524,Z 464.311,A -85,B 0,C 180,E1 -6555.876,E2 -6555.876} C_VEL
LIN {X 0,Y 490.128,Z 476.976,A -85,B 0,C 180,E1 -6556.42,E2 -6556.42} C_VEL
LIN {X 0,Y 489.732,Z 488.395,A -85,B 0,C 180,E1 -6557.074,E2 -6557.074} C_VEL
LIN {X 0,Y 489.425,Z 498.921,A -85,B 0,C 180,E1 -6557.833,E2 -6557.833} C_VEL
LIN {X 0,Y 488.952,Z 509.894,A -85,B 0,C 180,E1 -6558.811,E2 -6558.811} C_VEL
LIN {X 0,Y 488.644,Z 519.343,A -85,B 0,C 180,E1 -6559.852,E2 -6559.852} C_VEL
LIN {X 0,Y 488.399,Z 528.514,A -85,B 0,C 180,E1 -6561.101,E2 -6561.101} C_VEL
LIN {X 0,Y 488.244,Z 535.914,A -85,B 0,C 180,E1 -6562.348,E2 -6562.348} C_VEL
LIN {X 0,Y 488.158,Z 542.223,A -85,B 0,C 180,E1 -6563.686,E2 -6563.686} C_VEL
LIN {X 0,Y 488.1,Z 547.146,A -85,B 0,C 180,E1 -6565.044,E2 -6565.044} C_VEL
LIN {X 0,Y 488.145,Z 549.504,A -85,B 0,C 180,E1 -6565.872,E2 -6565.872} C_VEL
LIN {X 0,Y 488.099,Z 551.404,A -85,B 0,C 180,E1 -6566.698,E2 -6566.698} C_VEL
LIN {X 0,Y 488.084,Z 552.835,A -85,B 0,C 180,E1 -6567.524,E2 -6567.524} C_VEL
LIN {X 0,Y 488.046,Z 553.839,A -85,B 0,C 180,E1 -6568.35,E2 -6568.35} C_VEL
LIN {X 0,Y 488.11,Z 554.63,A -85,B 0,C 180,E1 -6570,E2 -6570} C_VEL
LIN {X 0,Y 488.124,Z 554.378,A -85,B 0,C 180,E1 -6570.825,E2 -6570.825} C_VEL
LIN {X 0,Y 488.064,Z 553.704,A -85,B 0,C 180,E1 -6571.65,E2 -6571.65} C_VEL
LIN {X 0,Y 488.109,Z 552.623,A -85,B 0,C 180,E1 -6572.476,E2 -6572.476} C_VEL
LIN {X 0,Y 488.13,Z 551.118,A -85,B 0,C 180,E1 -6573.302,E2 -6573.302} C_VEL
LIN {X 0,Y 488.162,Z 547.986,A -85,B 0,C 180,E1 -6574.542,E2 -6574.542} C_VEL
LIN {X 0,Y 488.23,Z 542.61,A -85,B 0,C 180,E1 -6576.07,E2 -6576.07} C_VEL
LIN {X 0,Y 488.277,Z 536.203,A -85,B 0,C 180,E1 -6577.443,E2 -6577.443} C_VEL
LIN {X 0,Y 488.431,Z 528.892,A -85,B 0,C 180,E1 -6578.69,E2 -6578.69} C_VEL
LIN {X 0,Y 488.617,Z 519.748,A -85,B 0,C 180,E1 -6579.939,E2 -6579.939} C_VEL
LIN {X 0,Y 488.956,Z 509.402,A -85,B 0,C 180,E1 -6581.084,E2 -6581.084} C_VEL
LIN {X 0,Y 489.304,Z 499.368,A -85,B 0,C 180,E1 -6581.985,E2 -6581.985} C_VEL
LIN {X 0,Y 489.65,Z 487.996,A -85,B 0,C 180,E1 -6582.812,E2 -6582.812} C_VEL
LIN {X 0,Y 490.02,Z 475.508,A -85,B 0,C 180,E1 -6583.53,E2 -6583.53} C_VEL
LIN {X 0,Y 490.375,Z 462.186,A -85,B 0,C 180,E1 -6584.102,E2 -6584.102} C_VEL
LIN {X 0,Y 489.197,Z 452.03,A -85,B 0,C 180,E1 -6584.455,E2 -6584.455} C_VEL
LIN {X 0,Y 488.472,Z 441.123,A -85,B 0,C 180,E1 -6584.743,E2 -6584.743} C_VEL
LIN {X 0,Y 488.7,Z 425.235,A -85,B 0,C 180,E1 -6587.962,E2 -6587.962} C_VEL
LIN {X 0,Y 488.821,Z 410.065,A -85,B 0,C 180,E1 -6591.066,E2 -6591.066} C_VEL
LIN {X 0,Y 488.965,Z 395.07,A -85,B 0,C 180,E1 -6594.182,E2 -6594.182} C_VEL
LIN {X 0,Y 489.154,Z 381.728,A -85,B 0,C 180,E1 -6597.026,E2 -6597.026} C_VEL
LIN {X 0,Y 489.306,Z 368.536,A -85,B 0,C 180,E1 -6599.942,E2 -6599.942} C_VEL
LIN {X 0,Y 489.566,Z 357.211,A -85,B 0,C 180,E1 -6602.57,E2 -6602.57} C_VEL
LIN {X 0,Y 490.246,Z 345.199,A -85,B 0,C 180,E1 -6605.539,E2 -6605.539} C_VEL
LIN {X 0,Y 490.042,Z 341.41,A -85,B 0,C 180,E1 -6606.569,E2 -6606.569} C_VEL
LIN {X 0,Y 488.717,Z 334.614,A -85,B 0,C 180,E1 -6608.657,E2 -6608.657} C_VEL
LIN {X 0,Y 488.712,Z 334.612,A -85,B 0,C 180,E1 -6611.6,E2 -6611.6} C_VEL
LIN {X 0,Y 488.716,Z 334.611,A -85,B 0,C 180,E1 -6614.801,E2 -6614.801} C_VEL
LIN {X 0,Y 488.695,Z 334.613,A -85,B 0,C 180,E1 -6617.475,E2 -6617.475} C_VEL
LIN {X 0,Y 488.737,Z 334.606,A -85,B 0,C 180,E1 -6619.677,E2 -6619.677} C_VEL
LIN {X 0,Y 488.686,Z 334.615,A -85,B 0,C 180,E1 -6622.841,E2 -6622.841} C_VEL
LIN {X 0,Y 488.738,Z 334.609,A -85,B 0,C 180,E1 -6625.888,E2 -6625.888} C_VEL
LIN {X 0,Y 488.697,Z 334.612,A -85,B 0,C 180,E1 -6628.82,E2 -6628.82} C_VEL
LIN {X 0,Y 488.749,Z 334.604,A -85,B 0,C 180,E1 -6631.671,E2 -6631.671} C_VEL
LIN {X 0,Y 488.732,Z 334.608,A -85,B 0,C 180,E1 -6634.443,E2 -6634.443} C_VEL
LIN {X 0,Y 488.726,Z 334.61,A -85,B 0,C 180,E1 -6637.153,E2 -6637.153} C_VEL
LIN {X 0,Y 488.73,Z 334.61,A -85,B 0,C 180,E1 -6639.811,E2 -6639.811} C_VEL
LIN {X 0,Y 488.734,Z 334.609,A -85,B 0,C 180,E1 -6642.423,E2 -6642.423} C_VEL
LIN {X 0,Y 488.761,Z 334.611,A -85,B 0,C 180,E1 -6645.133,E2 -6645.133} C_VEL
LIN {X 0,Y 490.832,Z 342.557,A -85,B 0,C 180,E1 -6645.594,E2 -6645.594} C_VEL
LIN {X 0,Y 490.572,Z 354.529,A -85,B 0,C 180,E1 -6646.327,E2 -6646.327} C_VEL
LIN {X 0,Y 490.253,Z 365.93,A -85,B 0,C 180,E1 -6647.218,E2 -6647.218} C_VEL
LIN {X 0,Y 489.861,Z 375.933,A -85,B 0,C 180,E1 -6648.203,E2 -6648.203} C_VEL
LIN {X 0,Y 489.518,Z 384.549,A -85,B 0,C 180,E1 -6649.243,E2 -6649.243} C_VEL
LIN {X 0,Y 489.188,Z 392.919,A -85,B 0,C 180,E1 -6650.49,E2 -6650.49} C_VEL
LIN {X 0,Y 488.943,Z 399.552,A -85,B 0,C 180,E1 -6651.736,E2 -6651.736} C_VEL
LIN {X 0,Y 488.722,Z 404.405,A -85,B 0,C 180,E1 -6652.863,E2 -6652.863} C_VEL
LIN {X 0,Y 488.603,Z 408.928,A -85,B 0,C 180,E1 -6654.221,E2 -6654.221} C_VEL
LIN {X 0,Y 488.454,Z 411.091,A -85,B 0,C 180,E1 -6655.047,E2 -6655.047} C_VEL
LIN {X 0,Y 488.416,Z 412.796,A -85,B 0,C 180,E1 -6655.874,E2 -6655.874} C_VEL
LIN {X 0,Y 488.368,Z 414.055,A -85,B 0,C 180,E1 -6656.7,E2 -6656.7} C_VEL
LIN {X 0,Y 488.301,Z 415.417,A -85,B 0,C 180,E1 -6658.35,E2 -6658.35} C_VEL
LIN {X 0,Y 488.244,Z 415.5,A -85,B 0,C 180,E1 -6659.175,E2 -6659.175} C_VEL
LIN {X 0,Y 488.247,Z 414.46,A -85,B 0,C 180,E1 -6660.825,E2 -6660.825} C_VEL
LIN {X 0,Y 488.307,Z 413.363,A -85,B 0,C 180,E1 -6661.649,E2 -6661.649} C_VEL
LIN {X 0,Y 488.286,Z 411.842,A -85,B 0,C 180,E1 -6662.475,E2 -6662.475} C_VEL
LIN {X 0,Y 488.547,Z 408.738,A -85,B 0,C 180,E1 -6663.711,E2 -6663.711} C_VEL
LIN {X 0,Y 488.543,Z 404.63,A -85,B 0,C 180,E1 -6664.951,E2 -6664.951} C_VEL
LIN {X 0,Y 488.823,Z 398.315,A -85,B 0,C 180,E1 -6666.397,E2 -6666.397} C_VEL
LIN {X 0,Y 489.064,Z 391.463,A -85,B 0,C 180,E1 -6667.639,E2 -6667.639} C_VEL
LIN {X 0,Y 489.312,Z 382.903,A -85,B 0,C 180,E1 -6668.882,E2 -6668.882} C_VEL
LIN {X 0,Y 489.701,Z 374.104,A -85,B 0,C 180,E1 -6669.917,E2 -6669.917} C_VEL
LIN {X 0,Y 490.091,Z 363.299,A -85,B 0,C 180,E1 -6670.953,E2 -6670.953} C_VEL
LIN {X 0,Y 490.381,Z 352.783,A -85,B 0,C 180,E1 -6671.76,E2 -6671.76} C_VEL
LIN {X 0,Y 490.675,Z 342.258,A -85,B 0,C 180,E1 -6672.406,E2 -6672.406} C_VEL
LIN {X 0,Y 488.769,Z 334.602,A -85,B 0,C 180,E1 -6672.882,E2 -6672.882} C_VEL
LIN {X 0,Y 488.765,Z 334.602,A -85,B 0,C 180,E1 -6675.855,E2 -6675.855} C_VEL
LIN {X 0,Y 488.744,Z 334.606,A -85,B 0,C 180,E1 -6679.313,E2 -6679.313} C_VEL
LIN {X 0,Y 488.702,Z 334.608,A -85,B 0,C 180,E1 -6681.957,E2 -6681.957} C_VEL
LIN {X 0,Y 488.748,Z 334.604,A -85,B 0,C 180,E1 -6685.052,E2 -6685.052} C_VEL
LIN {X 0,Y 488.75,Z 334.604,A -85,B 0,C 180,E1 -6687.396,E2 -6687.396} C_VEL
LIN {X 0,Y 488.714,Z 334.608,A -85,B 0,C 180,E1 -6690.363,E2 -6690.363} C_VEL
LIN {X 0,Y 488.738,Z 334.606,A -85,B 0,C 180,E1 -6693.484,E2 -6693.484} C_VEL
LIN {X 0,Y 488.685,Z 334.61,A -85,B 0,C 180,E1 -6696.354,E2 -6696.354} C_VEL
LIN {X 0,Y 488.745,Z 334.603,A -85,B 0,C 180,E1 -6699.25,E2 -6699.25} C_VEL
LIN {X 0,Y 488.715,Z 334.608,A -85,B 0,C 180,E1 -6701.6,E2 -6701.6} C_VEL
LIN {X 0,Y 488.714,Z 334.607,A -85,B 0,C 180,E1 -6704.801,E2 -6704.801} C_VEL
LIN {X 0,Y 488.699,Z 334.612,A -85,B 0,C 180,E1 -6707.475,E2 -6707.475} C_VEL
LIN {X 0,Y 488.735,Z 334.605,A -85,B 0,C 180,E1 -6709.676,E2 -6709.676} C_VEL
LIN {X 0,Y 488.681,Z 334.615,A -85,B 0,C 180,E1 -6712.841,E2 -6712.841} C_VEL
LIN {X 0,Y 488.732,Z 334.606,A -85,B 0,C 180,E1 -6715.887,E2 -6715.887} C_VEL
LIN {X 0,Y 488.694,Z 334.61,A -85,B 0,C 180,E1 -6718.82,E2 -6718.82} C_VEL
LIN {X 0,Y 488.737,Z 334.606,A -85,B 0,C 180,E1 -6721.832,E2 -6721.832} C_VEL
LIN {X 0,Y 488.06,Z 334.689,A -85,B 0,C 180,E1 -6722.52,E2 -6722.52} C_VEL
LIN {X 0,Y 485.214,Z 335.046,A -85,B 0,C 180,E1 -6723.637,E2 -6723.637} C_VEL
LIN {X 0,Y 482.81,Z 335.345,A -85,B 0,C 180,E1 -6724.538,E2 -6724.538} C_VEL
LIN {X 0,Y 481.771,Z 335.474,A -85,B 0,C 180,E1 -6725.233,E2 -6725.233} C_VEL
LIN {X 0,Y 481.682,Z 335.483,A -85,B 0,C 180,E1 -6725.469,E2 -6725.469} C_VEL
LIN {X 0,Y 481.65,Z 335.492,A -85,B 0,C 180,E1 -6728.605,E2 -6728.605} C_VEL
LIN {X 0,Y 481.707,Z 335.478,A -85,B 0,C 180,E1 -6731.502,E2 -6731.502} C_VEL
LIN {X 0,Y 481.744,Z 335.475,A -85,B 0,C 180,E1 -6734.776,E2 -6734.776} C_VEL
LIN {X 0,Y 481.752,Z 335.475,A -85,B 0,C 180,E1 -6738.215,E2 -6738.215} C_VEL
LIN {X 0,Y 481.764,Z 335.474,A -85,B 0,C 180,E1 -6741.612,E2 -6741.612} C_VEL
LIN {X 0,Y 481.811,Z 335.469,A -85,B 0,C 180,E1 -6744.14,E2 -6744.14} C_VEL
LIN {X 0,Y 481.93,Z 335.452,A -85,B 0,C 180,E1 -6747.493,E2 -6747.493} C_VEL
LIN {X 0,Y 481.907,Z 335.454,A -85,B 0,C 180,E1 -6750.836,E2 -6750.836} C_VEL
LIN {X 0,Y 481.931,Z 335.452,A -85,B 0,C 180,E1 -6752.508,E2 -6752.508} C_VEL
LIN {X 0,Y 481.811,Z 335.468,A -85,B 0,C 180,E1 -6755.861,E2 -6755.861} C_VEL
LIN {X 0,Y 481.765,Z 335.476,A -85,B 0,C 180,E1 -6758.388,E2 -6758.388} C_VEL
LIN {X 0,Y 481.753,Z 335.476,A -85,B 0,C 180,E1 -6761.785,E2 -6761.785} C_VEL
LIN {X 0,Y 481.744,Z 335.475,A -85,B 0,C 180,E1 -6765.224,E2 -6765.224} C_VEL
LIN {X 0,Y 481.714,Z 335.478,A -85,B 0,C 180,E1 -6768.722,E2 -6768.722} C_VEL
LIN {X 0,Y 481.648,Z 335.491,A -85,B 0,C 180,E1 -6771.395,E2 -6771.395} C_VEL
LIN {X 0,Y 481.676,Z 335.485,A -85,B 0,C 180,E1 -6774.113,E2 -6774.113} C_VEL
LIN {X 0,Y 481.748,Z 335.475,A -85,B 0,C 180,E1 -6777.139,E2 -6777.139} C_VEL
LIN {X 0,Y 481.681,Z 335.487,A -85,B 0,C 180,E1 -6779.741,E2 -6779.741} C_VEL
LIN {X 0,Y 481.674,Z 335.483,A -85,B 0,C 180,E1 -6782.674,E2 -6782.674} C_VEL
LIN {X 0,Y 481.639,Z 335.489,A -85,B 0,C 180,E1 -6785.71,E2 -6785.71} C_VEL
LIN {X 0,Y 481.673,Z 335.488,A -85,B 0,C 180,E1 -6788.859,E2 -6788.859} C_VEL
LIN {X 0,Y 481.677,Z 335.487,A -85,B 0,C 180,E1 -6792.158,E2 -6792.158} C_VEL
LIN {X 0,Y 481.663,Z 335.488,A -85,B 0,C 180,E1 -6794.457,E2 -6794.457} C_VEL
LIN {X 0,Y 481.651,Z 335.489,A -85,B 0,C 180,E1 -6797.84,E2 -6797.84} C_VEL
LIN {X 0,Y 481.683,Z 335.483,A -85,B 0,C 180,E1 -6800.651,E2 -6800.651} C_VEL
LIN {X 0,Y 481.631,Z 335.491,A -85,B 0,C 180,E1 -6803.376,E2 -6803.376} C_VEL
LIN {X 0,Y 481.713,Z 335.481,A -85,B 0,C 180,E1 -6806.33,E2 -6806.33} C_VEL
LIN {X 0,Y 481.654,Z 335.487,A -85,B 0,C 180,E1 -6809.418,E2 -6809.418} C_VEL
LIN {X 0,Y 481.705,Z 335.483,A -85,B 0,C 180,E1 -6812.168,E2 -6812.168} C_VEL
LIN {X 0,Y 481.722,Z 335.48,A -85,B 0,C 180,E1 -6814.97,E2 -6814.97} C_VEL
LIN {X 0,Y 481.654,Z 335.486,A -85,B 0,C 180,E1 -6817.705,E2 -6817.705} C_VEL
LIN {X 0,Y 481.708,Z 335.481,A -85,B 0,C 180,E1 -6820.393,E2 -6820.393} C_VEL
LIN {X 0,Y 481.692,Z 335.482,A -85,B 0,C 180,E1 -6823.034,E2 -6823.034} C_VEL
LIN {X 0,Y 481.696,Z 335.484,A -85,B 0,C 180,E1 -6825.639,E2 -6825.639} C_VEL
LIN {X 0,Y 481.757,Z 335.476,A -85,B 0,C 180,E1 -6828.215,E2 -6828.215} C_VEL
LIN {X 0,Y 481.769,Z 335.474,A -85,B 0,C 180,E1 -6831.612,E2 -6831.612} C_VEL
LIN {X 0,Y 481.821,Z 335.465,A -85,B 0,C 180,E1 -6834.14,E2 -6834.14} C_VEL
LIN {X 0,Y 481.932,Z 335.45,A -85,B 0,C 180,E1 -6837.493,E2 -6837.493} C_VEL
LIN {X 0,Y 481.911,Z 335.455,A -85,B 0,C 180,E1 -6840.836,E2 -6840.836} C_VEL
LIN {X 0,Y 481.934,Z 335.453,A -85,B 0,C 180,E1 -6842.508,E2 -6842.508} C_VEL
LIN {X 0,Y 481.813,Z 335.469,A -85,B 0,C 180,E1 -6845.861,E2 -6845.861} C_VEL
LIN {X 0,Y 481.746,Z 335.476,A -85,B 0,C 180,E1 -6848.389,E2 -6848.389} C_VEL
LIN {X 0,Y 481.757,Z 335.473,A -85,B 0,C 180,E1 -6851.785,E2 -6851.785} C_VEL
LIN {X 0,Y 481.748,Z 335.473,A -85,B 0,C 180,E1 -6855.224,E2 -6855.224} C_VEL
LIN {X 0,Y 481.718,Z 335.478,A -85,B 0,C 180,E1 -6858.722,E2 -6858.722} C_VEL
LIN {X 0,Y 481.651,Z 335.49,A -85,B 0,C 180,E1 -6861.395,E2 -6861.395} C_VEL
LIN {X 0,Y 481.679,Z 335.484,A -85,B 0,C 180,E1 -6864.113,E2 -6864.113} C_VEL
LIN {X 0,Y 481.752,Z 335.476,A -85,B 0,C 180,E1 -6867.139,E2 -6867.139} C_VEL
LIN {X 0,Y 481.684,Z 335.484,A -85,B 0,C 180,E1 -6869.741,E2 -6869.741} C_VEL
LIN {X 0,Y 481.677,Z 335.482,A -85,B 0,C 180,E1 -6872.674,E2 -6872.674} C_VEL
LIN {X 0,Y 481.646,Z 335.492,A -85,B 0,C 180,E1 -6875.709,E2 -6875.709} C_VEL
LIN {X 0,Y 481.676,Z 335.486,A -85,B 0,C 180,E1 -6878.859,E2 -6878.859} C_VEL
LIN {X 0,Y 481.657,Z 335.487,A -85,B 0,C 180,E1 -6881.913,E2 -6881.913} C_VEL
LIN {X 0,Y 481.664,Z 335.49,A -85,B 0,C 180,E1 -6884.457,E2 -6884.457} C_VEL
LIN {X 0,Y 481.658,Z 335.49,A -85,B 0,C 180,E1 -6887.84,E2 -6887.84} C_VEL
LIN {X 0,Y 481.706,Z 335.631,A -85,B 0,C 180,E1 -6889.605,E2 -6889.605} C_VEL
LIN {X 0,Y 483.969,Z 346.942,A -85,B 0,C 180,E1 -6892.744,E2 -6892.744} C_VEL
LIN {X 0,Y 484.47,Z 351.622,A -85,B 0,C 180,E1 -6893.975,E2 -6893.975} C_VEL
LIN {X 0,Y 483.79,Z 363.862,A -85,B 0,C 180,E1 -6896.992,E2 -6896.992} C_VEL
LIN {X 0,Y 483.25,Z 375.879,A -85,B 0,C 180,E1 -6899.884,E2 -6899.884} C_VEL
LIN {X 0,Y 482.856,Z 388.683,A -85,B 0,C 180,E1 -6902.888,E2 -6902.888} C_VEL
LIN {X 0,Y 482.328,Z 403.673,A -85,B 0,C 180,E1 -6906.329,E2 -6906.329} C_VEL
LIN {X 0,Y 481.933,Z 418.888,A -85,B 0,C 180,E1 -6909.736,E2 -6909.736} C_VEL
LIN {X 0,Y 481.583,Z 433.888,A -85,B 0,C 180,E1 -6913.03,E2 -6913.03} C_VEL
LIN {X 0,Y 481.43,Z 443.378,A -85,B 0,C 180,E1 -6915.063,E2 -6915.063} C_VEL
LIN {X 0,Y 482.815,Z 457.637,A -85,B 0,C 180,E1 -6915.457,E2 -6915.457} C_VEL
LIN {X 0,Y 483.575,Z 465.352,A -85,B 0,C 180,E1 -6915.749,E2 -6915.749} C_VEL
LIN {X 0,Y 483.109,Z 477.881,A -85,B 0,C 180,E1 -6916.326,E2 -6916.326} C_VEL
LIN {X 0,Y 482.645,Z 490,A -85,B 0,C 180,E1 -6917.063,E2 -6917.063} C_VEL
LIN {X 0,Y 482.293,Z 501.453,A -85,B 0,C 180,E1 -6917.952,E2 -6917.952} C_VEL
LIN {X 0,Y 481.885,Z 510.908,A -85,B 0,C 180,E1 -6918.858,E2 -6918.858} C_VEL
LIN {X 0,Y 481.526,Z 519.984,A -85,B 0,C 180,E1 -6919.913,E2 -6919.913} C_VEL
LIN {X 0,Y 481.289,Z 528.884,A -85,B 0,C 180,E1 -6921.18,E2 -6921.18} C_VEL
LIN {X 0,Y 481.165,Z 536.007,A -85,B 0,C 180,E1 -6922.446,E2 -6922.446} C_VEL
LIN {X 0,Y 481.094,Z 541.583,A -85,B 0,C 180,E1 -6923.679,E2 -6923.679} C_VEL
LIN {X 0,Y 481.036,Z 546.171,A -85,B 0,C 180,E1 -6924.971,E2 -6924.971} C_VEL
LIN {X 0,Y 481.079,Z 548.527,A -85,B 0,C 180,E1 -6925.811,E2 -6925.811} C_VEL
LIN {X 0,Y 481.053,Z 550.43,A -85,B 0,C 180,E1 -6926.65,E2 -6926.65} C_VEL
LIN {X 0,Y 481.039,Z 551.861,A -85,B 0,C 180,E1 -6927.488,E2 -6927.488} C_VEL
LIN {X 0,Y 481.01,Z 552.858,A -85,B 0,C 180,E1 -6928.325,E2 -6928.325} C_VEL
LIN {X 0,Y 481.094,Z 553.641,A -85,B 0,C 180,E1 -6930,E2 -6930} C_VEL
LIN {X 0,Y 481.11,Z 553.382,A -85,B 0,C 180,E1 -6930.837,E2 -6930.837} C_VEL
LIN {X 0,Y 481.071,Z 551.594,A -85,B 0,C 180,E1 -6932.512,E2 -6932.512} C_VEL
LIN {X 0,Y 481.091,Z 550.075,A -85,B 0,C 180,E1 -6933.35,E2 -6933.35} C_VEL
LIN {X 0,Y 481.107,Z 546.915,A -85,B 0,C 180,E1 -6934.608,E2 -6934.608} C_VEL
LIN {X 0,Y 481.171,Z 541.666,A -85,B 0,C 180,E1 -6936.117,E2 -6936.117} C_VEL
LIN {X 0,Y 481.226,Z 535.045,A -85,B 0,C 180,E1 -6937.553,E2 -6937.553} C_VEL
LIN {X 0,Y 481.346,Z 527.682,A -85,B 0,C 180,E1 -6938.819,E2 -6938.819} C_VEL
LIN {X 0,Y 481.57,Z 518.483,A -85,B 0,C 180,E1 -6940.086,E2 -6940.086} C_VEL
LIN {X 0,Y 481.853,Z 508.082,A -85,B 0,C 180,E1 -6941.249,E2 -6941.249} C_VEL
LIN {X 0,Y 482.234,Z 497.42,A -85,B 0,C 180,E1 -6942.21,E2 -6942.21} C_VEL
LIN {X 0,Y 482.661,Z 485.957,A -85,B 0,C 180,E1 -6943.044,E2 -6943.044} C_VEL
LIN {X 0,Y 483.068,Z 474.096,A -85,B 0,C 180,E1 -6943.729,E2 -6943.729} C_VEL
LIN {X 0,Y 483.272,Z 462.199,A -85,B 0,C 180,E1 -6944.26,E2 -6944.26} C_VEL
LIN {X 0,Y 482.259,Z 452.522,A -85,B 0,C 180,E1 -6944.614,E2 -6944.614} C_VEL
LIN {X 0,Y 481.412,Z 439.866,A -85,B 0,C 180,E1 -6944.964,E2 -6944.964} C_VEL
LIN {X 0,Y 481.618,Z 424.431,A -85,B 0,C 180,E1 -6948.15,E2 -6948.15} C_VEL
LIN {X 0,Y 481.722,Z 410.85,A -85,B 0,C 180,E1 -6950.978,E2 -6950.978} C_VEL
LIN {X 0,Y 481.922,Z 396.1,A -85,B 0,C 180,E1 -6954.1,E2 -6954.1} C_VEL
LIN {X 0,Y 482.099,Z 381.752,A -85,B 0,C 180,E1 -6957.22,E2 -6957.22} C_VEL
LIN {X 0,Y 482.307,Z 368.674,A -85,B 0,C 180,E1 -6960.18,E2 -6960.18} C_VEL
LIN {X 0,Y 482.592,Z 358.469,A -85,B 0,C 180,E1 -6962.604,E2 -6962.604} C_VEL
LIN {X 0,Y 483.311,Z 346.768,A -85,B 0,C 180,E1 -6965.567,E2 -6965.567} C_VEL
LIN {X 0,Y 483.142,Z 343.004,A -85,B 0,C 180,E1 -6966.613,E2 -6966.613} C_VEL
LIN {X 0,Y 481.677,Z 335.49,A -85,B 0,C 180,E1 -6968.981,E2 -6968.981} C_VEL
LIN {X 0,Y 481.651,Z 335.49,A -85,B 0,C 180,E1 -6972.161,E2 -6972.161} C_VEL
LIN {X 0,Y 481.663,Z 335.489,A -85,B 0,C 180,E1 -6975.543,E2 -6975.543} C_VEL
LIN {X 0,Y 481.66,Z 335.488,A -85,B 0,C 180,E1 -6978.958,E2 -6978.958} C_VEL
LIN {X 0,Y 481.66,Z 335.487,A -85,B 0,C 180,E1 -6981.993,E2 -6981.993} C_VEL
LIN {X 0,Y 481.696,Z 335.484,A -85,B 0,C 180,E1 -6985.318,E2 -6985.318} C_VEL
LIN {X 0,Y 481.65,Z 335.491,A -85,B 0,C 180,E1 -6988.312,E2 -6988.312} C_VEL
LIN {X 0,Y 481.705,Z 335.484,A -85,B 0,C 180,E1 -6991.219,E2 -6991.219} C_VEL
LIN {X 0,Y 481.694,Z 335.485,A -85,B 0,C 180,E1 -6994.042,E2 -6994.042} C_VEL
LIN {X 0,Y 481.678,Z 335.487,A -85,B 0,C 180,E1 -6996.812,E2 -6996.812} C_VEL
LIN {X 0,Y 481.7,Z 335.486,A -85,B 0,C 180,E1 -6999.503,E2 -6999.503} C_VEL
LIN {X 0,Y 481.709,Z 335.484,A -85,B 0,C 180,E1 -7002.158,E2 -7002.158} C_VEL
LIN {X 0,Y 481.726,Z 335.482,A -85,B 0,C 180,E1 -7004.883,E2 -7004.883} C_VEL
LIN {X 0,Y 483.917,Z 343.494,A -85,B 0,C 180,E1 -7005.384,E2 -7005.384} C_VEL
LIN {X 0,Y 483.734,Z 355.422,A -85,B 0,C 180,E1 -7006.13,E2 -7006.13} C_VEL
LIN {X 0,Y 483.401,Z 366.819,A -85,B 0,C 180,E1 -7007.034,E2 -7007.034} C_VEL
LIN {X 0,Y 482.973,Z 376.854,A -85,B 0,C 180,E1 -7008.032,E2 -7008.032} C_VEL
LIN {X 0,Y 482.612,Z 385.496,A -85,B 0,C 180,E1 -7009.087,E2 -7009.087} C_VEL
LIN {X 0,Y 482.255,Z 393.901,A -85,B 0,C 180,E1 -7010.352,E2 -7010.352} C_VEL
LIN {X 0,Y 481.989,Z 400.554,A -85,B 0,C 180,E1 -7011.616,E2 -7011.616} C_VEL
LIN {X 0,Y 481.749,Z 405.42,A -85,B 0,C 180,E1 -7012.759,E2 -7012.759} C_VEL
LIN {X 0,Y 481.638,Z 409.95,A -85,B 0,C 180,E1 -7014.137,E2 -7014.137} C_VEL
LIN {X 0,Y 481.453,Z 412.117,A -85,B 0,C 180,E1 -7014.975,E2 -7014.975} C_VEL
LIN {X 0,Y 481.406,Z 413.827,A -85,B 0,C 180,E1 -7015.814,E2 -7015.814} C_VEL
LIN {X 0,Y 481.352,Z 415.084,A -85,B 0,C 180,E1 -7016.652,E2 -7016.652} C_VEL
LIN {X 0,Y 481.285,Z 416.436,A -85,B 0,C 180,E1 -7018.326,E2 -7018.326} C_VEL
LIN {X 0,Y 481.224,Z 416.516,A -85,B 0,C 180,E1 -7019.163,E2 -7019.163} C_VEL
LIN {X 0,Y 481.226,Z 415.466,A -85,B 0,C 180,E1 -7020.837,E2 -7020.837} C_VEL
LIN {X 0,Y 481.291,Z 414.359,A -85,B 0,C 180,E1 -7021.673,E2 -7021.673} C_VEL
LIN {X 0,Y 481.262,Z 412.83,A -85,B 0,C 180,E1 -7022.511,E2 -7022.511} C_VEL
LIN {X 0,Y 481.536,Z 409.71,A -85,B 0,C 180,E1 -7023.766,E2 -7023.766} C_VEL
LIN {X 0,Y 481.534,Z 405.585,A -85,B 0,C 180,E1 -7025.024,E2 -7025.024} C_VEL
LIN {X 0,Y 481.837,Z 399.251,A -85,B 0,C 180,E1 -7026.49,E2 -7026.49} C_VEL
LIN {X 0,Y 482.099,Z 392.376,A -85,B 0,C 180,E1 -7027.75,E2 -7027.75} C_VEL
LIN {X 0,Y 482.369,Z 383.787,A -85,B 0,C 180,E1 -7029.011,E2 -7029.011} C_VEL
LIN {X 0,Y 482.779,Z 374.968,A -85,B 0,C 180,E1 -7030.06,E2 -7030.06} C_VEL
LIN {X 0,Y 483.183,Z 364.137,A -85,B 0,C 180,E1 -7031.112,E2 -7031.112} C_VEL
LIN {X 0,Y 483.49,Z 353.719,A -85,B 0,C 180,E1 -7031.921,E2 -7031.921} C_VEL
LIN {X 0,Y 483.775,Z 343.068,A -85,B 0,C 180,E1 -7032.586,E2 -7032.586} C_VEL
LIN {X 0,Y 481.711,Z 335.481,A -85,B 0,C 180,E1 -7033.056,E2 -7033.056} C_VEL
LIN {X 0,Y 481.698,Z 335.481,A -85,B 0,C 180,E1 -7036.094,E2 -7036.094} C_VEL
LIN {X 0,Y 481.711,Z 335.48,A -85,B 0,C 180,E1 -7038.722,E2 -7038.722} C_VEL
LIN {X 0,Y 481.649,Z 335.488,A -85,B 0,C 180,E1 -7041.394,E2 -7041.394} C_VEL
LIN {X 0,Y 481.678,Z 335.486,A -85,B 0,C 180,E1 -7044.113,E2 -7044.113} C_VEL
LIN {X 0,Y 481.751,Z 335.475,A -85,B 0,C 180,E1 -7047.139,E2 -7047.139} C_VEL
LIN {X 0,Y 481.683,Z 335.486,A -85,B 0,C 180,E1 -7049.741,E2 -7049.741} C_VEL
LIN {X 0,Y 481.676,Z 335.484,A -85,B 0,C 180,E1 -7052.674,E2 -7052.674} C_VEL
LIN {X 0,Y 481.64,Z 335.487,A -85,B 0,C 180,E1 -7055.709,E2 -7055.709} C_VEL
LIN {X 0,Y 481.717,Z 335.478,A -85,B 0,C 180,E1 -7059.354,E2 -7059.354} C_VEL
LIN {X 0,Y 481.651,Z 335.49,A -85,B 0,C 180,E1 -7062.16,E2 -7062.16} C_VEL
LIN {X 0,Y 481.663,Z 335.489,A -85,B 0,C 180,E1 -7065.543,E2 -7065.543} C_VEL
LIN {X 0,Y 481.665,Z 335.486,A -85,B 0,C 180,E1 -7068.086,E2 -7068.086} C_VEL
LIN {X 0,Y 481.673,Z 335.486,A -85,B 0,C 180,E1 -7071.141,E2 -7071.141} C_VEL
LIN {X 0,Y 481.664,Z 335.487,A -85,B 0,C 180,E1 -7074.796,E2 -7074.796} C_VEL
LIN {X 0,Y 481.674,Z 335.484,A -85,B 0,C 180,E1 -7077.326,E2 -7077.326} C_VEL
LIN {X 0,Y 481.68,Z 335.485,A -85,B 0,C 180,E1 -7080.259,E2 -7080.259} C_VEL
LIN {X 0,Y 481.747,Z 335.479,A -85,B 0,C 180,E1 -7083.112,E2 -7083.112} C_VEL
LIN {X 0,Y 481.682,Z 335.483,A -85,B 0,C 180,E1 -7085.469,E2 -7085.469} C_VEL
LIN {X 0,Y 480.992,Z 335.57,A -85,B 0,C 180,E1 -7086.166,E2 -7086.166} C_VEL
LIN {X 0,Y 478.099,Z 335.931,A -85,B 0,C 180,E1 -7087.298,E2 -7087.298} C_VEL
LIN {X 0,Y 475.699,Z 336.23,A -85,B 0,C 180,E1 -7088.21,E2 -7088.21} C_VEL
LIN {X 0,Y 474.721,Z 336.352,A -85,B 0,C 180,E1 -7088.916,E2 -7088.916} C_VEL
LIN {X 0,Y 474.668,Z 336.357,A -85,B 0,C 180,E1 -7089.154,E2 -7089.154} C_VEL
LIN {X 0,Y 474.659,Z 336.359,A -85,B 0,C 180,E1 -7091.884,E2 -7091.884} C_VEL
LIN {X 0,Y 474.701,Z 336.353,A -85,B 0,C 180,E1 -7094.544,E2 -7094.544} C_VEL
LIN {X 0,Y 474.706,Z 336.354,A -85,B 0,C 180,E1 -7098.038,E2 -7098.038} C_VEL
LIN {X 0,Y 474.729,Z 336.351,A -85,B 0,C 180,E1 -7101.486,E2 -7101.486} C_VEL
LIN {X 0,Y 474.773,Z 336.345,A -85,B 0,C 180,E1 -7104.052,E2 -7104.052} C_VEL
LIN {X 0,Y 474.896,Z 336.328,A -85,B 0,C 180,E1 -7107.455,E2 -7107.455} C_VEL
LIN {X 0,Y 474.913,Z 336.331,A -85,B 0,C 180,E1 -7110,E2 -7110} C_VEL
LIN {X 0,Y 474.897,Z 336.328,A -85,B 0,C 180,E1 -7112.545,E2 -7112.545} C_VEL
LIN {X 0,Y 474.773,Z 336.344,A -85,B 0,C 180,E1 -7115.948,E2 -7115.948} C_VEL
LIN {X 0,Y 474.73,Z 336.353,A -85,B 0,C 180,E1 -7118.514,E2 -7118.514} C_VEL
LIN {X 0,Y 474.706,Z 336.355,A -85,B 0,C 180,E1 -7121.963,E2 -7121.963} C_VEL
LIN {X 0,Y 474.702,Z 336.354,A -85,B 0,C 180,E1 -7125.456,E2 -7125.456} C_VEL
LIN {X 0,Y 474.667,Z 336.358,A -85,B 0,C 180,E1 -7129.01,E2 -7129.01} C_VEL
LIN {X 0,Y 474.59,Z 336.367,A -85,B 0,C 180,E1 -7131.729,E2 -7131.729} C_VEL
LIN {X 0,Y 474.659,Z 336.361,A -85,B 0,C 180,E1 -7134.493,E2 -7134.493} C_VEL
LIN {X 0,Y 474.683,Z 336.355,A -85,B 0,C 180,E1 -7137.335,E2 -7137.335} C_VEL
LIN {X 0,Y 474.607,Z 336.366,A -85,B 0,C 180,E1 -7140.23,E2 -7140.23} C_VEL
LIN {X 0,Y 474.645,Z 336.362,A -85,B 0,C 180,E1 -7143.22,E2 -7143.22} C_VEL
LIN {X 0,Y 474.591,Z 336.366,A -85,B 0,C 180,E1 -7146.324,E2 -7146.324} C_VEL
LIN {X 0,Y 474.63,Z 336.362,A -85,B 0,C 180,E1 -7149.648,E2 -7149.648} C_VEL
LIN {X 0,Y 474.655,Z 336.36,A -85,B 0,C 180,E1 -7152.93,E2 -7152.93} C_VEL
LIN {X 0,Y 474.612,Z 336.367,A -85,B 0,C 180,E1 -7155.896,E2 -7155.896} C_VEL
LIN {X 0,Y 474.631,Z 336.363,A -85,B 0,C 180,E1 -7159.041,E2 -7159.041} C_VEL
LIN {X 0,Y 474.613,Z 336.363,A -85,B 0,C 180,E1 -7161.704,E2 -7161.704} C_VEL
LIN {X 0,Y 474.629,Z 336.365,A -85,B 0,C 180,E1 -7164.726,E2 -7164.726} C_VEL
LIN {X 0,Y 474.639,Z 336.362,A -85,B 0,C 180,E1 -7167.788,E2 -7167.788} C_VEL
LIN {X 0,Y 474.628,Z 336.362,A -85,B 0,C 180,E1 -7170.885,E2 -7170.885} C_VEL
LIN {X 0,Y 474.665,Z 336.36,A -85,B 0,C 180,E1 -7173.629,E2 -7173.629} C_VEL
LIN {X 0,Y 474.64,Z 336.361,A -85,B 0,C 180,E1 -7176.642,E2 -7176.642} C_VEL
LIN {X 0,Y 474.658,Z 336.357,A -85,B 0,C 180,E1 -7180.09,E2 -7180.09} C_VEL
LIN {X 0,Y 474.652,Z 336.361,A -85,B 0,C 180,E1 -7182.775,E2 -7182.775} C_VEL
LIN {X 0,Y 474.654,Z 336.36,A -85,B 0,C 180,E1 -7185.421,E2 -7185.421} C_VEL
LIN {X 0,Y 474.71,Z 336.355,A -85,B 0,C 180,E1 -7188.038,E2 -7188.038} C_VEL
LIN {X 0,Y 474.734,Z 336.351,A -85,B 0,C 180,E1 -7191.487,E2 -7191.487} C_VEL
LIN {X 0,Y 474.784,Z 336.342,A -85,B 0,C 180,E1 -7194.053,E2 -7194.053} C_VEL
LIN {X 0,Y 474.898,Z 336.326,A -85,B 0,C 180,E1 -7197.456,E2 -7197.456} C_VEL
LIN {X 0,Y 474.918,Z 336.328,A -85,B 0,C 180,E1 -7200,E2 -7200} C_VEL
LIN {X 0,Y 474.9,Z 336.329,A -85,B 0,C 180,E1 -7202.545,E2 -7202.545} C_VEL
LIN {X 0,Y 474.775,Z 336.346,A -85,B 0,C 180,E1 -7205.948,E2 -7205.948} C_VEL
LIN {X 0,Y 474.717,Z 336.353,A -85,B 0,C 180,E1 -7208.514,E2 -7208.514} C_VEL
LIN {X 0,Y 474.71,Z 336.352,A -85,B 0,C 180,E1 -7211.962,E2 -7211.962} C_VEL
LIN {X 0,Y 474.706,Z 336.351,A -85,B 0,C 180,E1 -7215.456,E2 -7215.456} C_VEL
LIN {X 0,Y 474.672,Z 336.357,A -85,B 0,C 180,E1 -7219.01,E2 -7219.01} C_VEL
LIN {X 0,Y 474.594,Z 336.369,A -85,B 0,C 180,E1 -7221.729,E2 -7221.729} C_VEL
LIN {X 0,Y 474.662,Z 336.36,A -85,B 0,C 180,E1 -7224.493,E2 -7224.493} C_VEL
LIN {X 0,Y 474.686,Z 336.355,A -85,B 0,C 180,E1 -7227.334,E2 -7227.334} C_VEL
LIN {X 0,Y 474.611,Z 336.368,A -85,B 0,C 180,E1 -7230.23,E2 -7230.23} C_VEL
LIN {X 0,Y 474.648,Z 336.358,A -85,B 0,C 180,E1 -7233.22,E2 -7233.22} C_VEL
LIN {X 0,Y 474.597,Z 336.366,A -85,B 0,C 180,E1 -7236.323,E2 -7236.323} C_VEL
LIN {X 0,Y 474.632,Z 336.363,A -85,B 0,C 180,E1 -7239.648,E2 -7239.648} C_VEL
LIN {X 0,Y 474.619,Z 336.366,A -85,B 0,C 180,E1 -7242.934,E2 -7242.934} C_VEL
LIN {X 0,Y 474.62,Z 336.366,A -85,B 0,C 180,E1 -7245.896,E2 -7245.896} C_VEL
LIN {X 0,Y 474.635,Z 336.364,A -85,B 0,C 180,E1 -7249.192,E2 -7249.192} C_VEL
LIN {X 0,Y 474.67,Z 336.605,A -85,B 0,C 180,E1 -7249.347,E2 -7249.347} C_VEL
LIN {X 0,Y 476.765,Z 346.932,A -85,B 0,C 180,E1 -7252.268,E2 -7252.268} C_VEL
LIN {X 0,Y 477.524,Z 352.133,A -85,B 0,C 180,E1 -7253.673,E2 -7253.673} C_VEL
LIN {X 0,Y 476.938,Z 363.172,A -85,B 0,C 180,E1 -7256.455,E2 -7256.455} C_VEL
LIN {X 0,Y 476.37,Z 375.213,A -85,B 0,C 180,E1 -7259.403,E2 -7259.403} C_VEL
LIN {X 0,Y 475.846,Z 389.21,A -85,B 0,C 180,E1 -7262.751,E2 -7262.751} C_VEL
LIN {X 0,Y 475.264,Z 405.183,A -85,B 0,C 180,E1 -7266.468,E2 -7266.468} C_VEL
LIN {X 0,Y 474.838,Z 420.1,A -85,B 0,C 180,E1 -7269.872,E2 -7269.872} C_VEL
LIN {X 0,Y 474.522,Z 433.021,A -85,B 0,C 180,E1 -7272.769,E2 -7272.769} C_VEL
LIN {X 0,Y 474.345,Z 442.328,A -85,B 0,C 180,E1 -7274.835,E2 -7274.835} C_VEL
LIN {X 0,Y 475.762,Z 457.336,A -85,B 0,C 180,E1 -7275.264,E2 -7275.264} C_VEL
LIN {X 0,Y 476.62,Z 465.539,A -85,B 0,C 180,E1 -7275.592,E2 -7275.592} C_VEL
LIN {X 0,Y 476.164,Z 476.803,A -85,B 0,C 180,E1 -7276.123,E2 -7276.123} C_VEL
LIN {X 0,Y 475.682,Z 488.94,A -85,B 0,C 180,E1 -7276.87,E2 -7276.87} C_VEL
LIN {X 0,Y 475.32,Z 499.965,A -85,B 0,C 180,E1 -7277.732,E2 -7277.732} C_VEL
LIN {X 0,Y 474.791,Z 509.873,A -85,B 0,C 180,E1 -7278.689,E2 -7278.689} C_VEL
LIN {X 0,Y 474.481,Z 518.971,A -85,B 0,C 180,E1 -7279.761,E2 -7279.761} C_VEL
LIN {X 0,Y 474.23,Z 527.884,A -85,B 0,C 180,E1 -7281.048,E2 -7281.048} C_VEL
LIN {X 0,Y 474.089,Z 535.02,A -85,B 0,C 180,E1 -7282.333,E2 -7282.333} C_VEL
LIN {X 0,Y 474.03,Z 540.939,A -85,B 0,C 180,E1 -7283.671,E2 -7283.671} C_VEL
LIN {X 0,Y 473.974,Z 545.193,A -85,B 0,C 180,E1 -7284.896,E2 -7284.896} C_VEL
LIN {X 0,Y 474.018,Z 547.551,A -85,B 0,C 180,E1 -7285.749,E2 -7285.749} C_VEL
LIN {X 0,Y 474.007,Z 549.456,A -85,B 0,C 180,E1 -7286.6,E2 -7286.6} C_VEL
LIN {X 0,Y 473.993,Z 550.887,A -85,B 0,C 180,E1 -7287.45,E2 -7287.45} C_VEL
LIN {X 0,Y 473.972,Z 551.876,A -85,B 0,C 180,E1 -7288.301,E2 -7288.301} C_VEL
LIN {X 0,Y 474.077,Z 552.652,A -85,B 0,C 180,E1 -7290,E2 -7290} C_VEL
LIN {X 0,Y 474.094,Z 552.383,A -85,B 0,C 180,E1 -7290.849,E2 -7290.849} C_VEL
LIN {X 0,Y 474.032,Z 550.565,A -85,B 0,C 180,E1 -7292.549,E2 -7292.549} C_VEL
LIN {X 0,Y 474.084,Z 548.07,A -85,B 0,C 180,E1 -7293.825,E2 -7293.825} C_VEL
LIN {X 0,Y 474.085,Z 544.519,A -85,B 0,C 180,E1 -7295.103,E2 -7295.103} C_VEL
LIN {X 0,Y 474.09,Z 539.784,A -85,B 0,C 180,E1 -7296.395,E2 -7296.395} C_VEL
LIN {X 0,Y 474.17,Z 533.892,A -85,B 0,C 180,E1 -7297.666,E2 -7297.666} C_VEL
LIN {X 0,Y 474.275,Z 526.482,A -85,B 0,C 180,E1 -7298.951,E2 -7298.951} C_VEL
LIN {X 0,Y 474.507,Z 517.241,A -85,B 0,C 180,E1 -7300.238,E2 -7300.238} C_VEL
LIN {X 0,Y 474.82,Z 506.792,A -85,B 0,C 180,E1 -7301.418,E2 -7301.418} C_VEL
LIN {X 0,Y 475.167,Z 498.104,A -85,B 0,C 180,E1 -7302.226,E2 -7302.226} C_VEL
LIN {X 0,Y 475.623,Z 486.247,A -85,B 0,C 180,E1 -7303.132,E2 -7303.132} C_VEL
LIN {X 0,Y 476.072,Z 473.792,A -85,B 0,C 180,E1 -7303.88,E2 -7303.88} C_VEL
LIN {X 0,Y 476.347,Z 463.542,A -85,B 0,C 180,E1 -7304.362,E2 -7304.362} C_VEL
LIN {X 0,Y 475.317,Z 453.103,A -85,B 0,C 180,E1 -7304.777,E2 -7304.777} C_VEL
LIN {X 0,Y 474.354,Z 438.632,A -85,B 0,C 180,E1 -7305.192,E2 -7305.192} C_VEL
LIN {X 0,Y 474.511,Z 423.626,A -85,B 0,C 180,E1 -7308.344,E2 -7308.344} C_VEL
LIN {X 0,Y 474.658,Z 409.351,A -85,B 0,C 180,E1 -7311.377,E2 -7311.377} C_VEL
LIN {X 0,Y 474.862,Z 394.997,A -85,B 0,C 180,E1 -7314.482,E2 -7314.482} C_VEL
LIN {X 0,Y 475.07,Z 381.79,A -85,B 0,C 180,E1 -7317.424,E2 -7317.424} C_VEL
LIN {X 0,Y 475.359,Z 368.204,A -85,B 0,C 180,E1 -7320.578,E2 -7320.578} C_VEL
LIN {X 0,Y 475.686,Z 357.765,A -85,B 0,C 180,E1 -7323.138,E2 -7323.138} C_VEL
LIN {X 0,Y 476.395,Z 347.702,A -85,B 0,C 180,E1 -7325.768,E2 -7325.768} C_VEL
LIN {X 0,Y 476.266,Z 344.682,A -85,B 0,C 180,E1 -7326.632,E2 -7326.632} C_VEL
LIN {X 0,Y 474.664,Z 336.364,A -85,B 0,C 180,E1 -7329.338,E2 -7329.338} C_VEL
LIN {X 0,Y 474.628,Z 336.365,A -85,B 0,C 180,E1 -7332.237,E2 -7332.237} C_VEL
LIN {X 0,Y 474.625,Z 336.365,A -85,B 0,C 180,E1 -7335.297,E2 -7335.297} C_VEL
LIN {X 0,Y 474.624,Z 336.364,A -85,B 0,C 180,E1 -7338.215,E2 -7338.215} C_VEL
LIN {X 0,Y 474.648,Z 336.361,A -85,B 0,C 180,E1 -7340.454,E2 -7340.454} C_VEL
LIN {X 0,Y 474.596,Z 336.367,A -85,B 0,C 180,E1 -7343.677,E2 -7343.677} C_VEL
LIN {X 0,Y 474.647,Z 336.363,A -85,B 0,C 180,E1 -7346.78,E2 -7346.78} C_VEL
LIN {X 0,Y 474.61,Z 336.368,A -85,B 0,C 180,E1 -7349.77,E2 -7349.77} C_VEL
LIN {X 0,Y 474.701,Z 336.357,A -85,B 0,C 180,E1 -7352.68,E2 -7352.68} C_VEL
LIN {X 0,Y 474.645,Z 336.363,A -85,B 0,C 180,E1 -7355.506,E2 -7355.506} C_VEL
LIN {X 0,Y 474.675,Z 336.36,A -85,B 0,C 180,E1 -7359.185,E2 -7359.185} C_VEL
LIN {X 0,Y 474.66,Z 336.361,A -85,B 0,C 180,E1 -7361.884,E2 -7361.884} C_VEL
LIN {X 0,Y 474.711,Z 336.356,A -85,B 0,C 180,E1 -7364.655,E2 -7364.655} C_VEL
LIN {X 0,Y 477.011,Z 344.557,A -85,B 0,C 180,E1 -7365.167,E2 -7365.167} C_VEL
LIN {X 0,Y 477.097,Z 351.711,A -85,B 0,C 180,E1 -7365.606,E2 -7365.606} C_VEL
LIN {X 0,Y 476.732,Z 363.277,A -85,B 0,C 180,E1 -7366.448,E2 -7366.448} C_VEL
LIN {X 0,Y 476.294,Z 373.906,A -85,B 0,C 180,E1 -7367.429,E2 -7367.429} C_VEL
LIN {X 0,Y 475.914,Z 383.271,A -85,B 0,C 180,E1 -7368.5,E2 -7368.5} C_VEL
LIN {X 0,Y 475.547,Z 390.939,A -85,B 0,C 180,E1 -7369.569,E2 -7369.569} C_VEL
LIN {X 0,Y 475.198,Z 398.413,A -85,B 0,C 180,E1 -7370.852,E2 -7370.852} C_VEL
LIN {X 0,Y 474.838,Z 405.237,A -85,B 0,C 180,E1 -7372.345,E2 -7372.345} C_VEL
LIN {X 0,Y 474.735,Z 409.725,A -85,B 0,C 180,E1 -7373.625,E2 -7373.625} C_VEL
LIN {X 0,Y 474.454,Z 413.142,A -85,B 0,C 180,E1 -7374.901,E2 -7374.901} C_VEL
LIN {X 0,Y 474.396,Z 414.858,A -85,B 0,C 180,E1 -7375.752,E2 -7375.752} C_VEL
LIN {X 0,Y 474.337,Z 416.117,A -85,B 0,C 180,E1 -7376.602,E2 -7376.602} C_VEL
LIN {X 0,Y 474.268,Z 417.459,A -85,B 0,C 180,E1 -7378.302,E2 -7378.302} C_VEL
LIN {X 0,Y 474.202,Z 417.538,A -85,B 0,C 180,E1 -7379.151,E2 -7379.151} C_VEL
LIN {X 0,Y 474.205,Z 416.472,A -85,B 0,C 180,E1 -7380.849,E2 -7380.849} C_VEL
LIN {X 0,Y 474.273,Z 415.353,A -85,B 0,C 180,E1 -7381.698,E2 -7381.698} C_VEL
LIN {X 0,Y 474.239,Z 413.817,A -85,B 0,C 180,E1 -7382.548,E2 -7382.548} C_VEL
LIN {X 0,Y 474.525,Z 410.678,A -85,B 0,C 180,E1 -7383.821,E2 -7383.821} C_VEL
LIN {X 0,Y 474.527,Z 406.533,A -85,B 0,C 180,E1 -7385.098,E2 -7385.098} C_VEL
LIN {X 0,Y 474.853,Z 400.171,A -85,B 0,C 180,E1 -7386.586,E2 -7386.586} C_VEL
LIN {X 0,Y 475.137,Z 393.267,A -85,B 0,C 180,E1 -7387.864,E2 -7387.864} C_VEL
LIN {X 0,Y 475.43,Z 384.65,A -85,B 0,C 180,E1 -7389.144,E2 -7389.144} C_VEL
LIN {X 0,Y 475.862,Z 375.806,A -85,B 0,C 180,E1 -7390.208,E2 -7390.208} C_VEL
LIN {X 0,Y 476.278,Z 364.946,A -85,B 0,C 180,E1 -7391.275,E2 -7391.275} C_VEL
LIN {X 0,Y 476.585,Z 354.625,A -85,B 0,C 180,E1 -7392.088,E2 -7392.088} C_VEL
LIN {X 0,Y 476.924,Z 345.599,A -85,B 0,C 180,E1 -7392.67,E2 -7392.67} C_VEL
LIN {X 0,Y 475.366,Z 338.959,A -85,B 0,C 180,E1 -7393.086,E2 -7393.086} C_VEL
LIN {X 0,Y 474.662,Z 336.361,A -85,B 0,C 180,E1 -7393.254,E2 -7393.254} C_VEL
LIN {X 0,Y 474.643,Z 336.359,A -85,B 0,C 180,E1 -7396.34,E2 -7396.34} C_VEL
LIN {X 0,Y 474.666,Z 336.361,A -85,B 0,C 180,E1 -7399.01,E2 -7399.01} C_VEL
LIN {X 0,Y 474.592,Z 336.366,A -85,B 0,C 180,E1 -7401.729,E2 -7401.729} C_VEL
LIN {X 0,Y 474.661,Z 336.361,A -85,B 0,C 180,E1 -7404.493,E2 -7404.493} C_VEL
LIN {X 0,Y 474.703,Z 336.354,A -85,B 0,C 180,E1 -7407.338,E2 -7407.338} C_VEL
LIN {X 0,Y 474.608,Z 336.365,A -85,B 0,C 180,E1 -7410.81,E2 -7410.81} C_VEL
LIN {X 0,Y 474.64,Z 336.359,A -85,B 0,C 180,E1 -7413.984,E2 -7413.984} C_VEL
LIN {X 0,Y 474.575,Z 336.373,A -85,B 0,C 180,E1 -7416.899,E2 -7416.899} C_VEL
LIN {X 0,Y 474.653,Z 336.359,A -85,B 0,C 180,E1 -7419.651,E2 -7419.651} C_VEL
LIN {X 0,Y 474.617,Z 336.364,A -85,B 0,C 180,E1 -7422.934,E2 -7422.934} C_VEL
LIN {X 0,Y 474.62,Z 336.366,A -85,B 0,C 180,E1 -7425.896,E2 -7425.896} C_VEL
LIN {X 0,Y 474.634,Z 336.366,A -85,B 0,C 180,E1 -7429.04,E2 -7429.04} C_VEL
LIN {X 0,Y 474.611,Z 336.363,A -85,B 0,C 180,E1 -7431.704,E2 -7431.704} C_VEL
LIN {X 0,Y 474.626,Z 336.365,A -85,B 0,C 180,E1 -7434.726,E2 -7434.726} C_VEL
LIN {X 0,Y 474.638,Z 336.362,A -85,B 0,C 180,E1 -7437.788,E2 -7437.788} C_VEL
LIN {X 0,Y 474.626,Z 336.363,A -85,B 0,C 180,E1 -7440.884,E2 -7440.884} C_VEL
LIN {X 0,Y 474.662,Z 336.36,A -85,B 0,C 180,E1 -7443.628,E2 -7443.628} C_VEL
LIN {X 0,Y 474.637,Z 336.365,A -85,B 0,C 180,E1 -7446.641,E2 -7446.641} C_VEL
LIN {X 0,Y 474.668,Z 336.357,A -85,B 0,C 180,E1 -7449.154,E2 -7449.154} C_VEL
LIN {X 0,Y 474.068,Z 336.433,A -85,B 0,C 180,E1 -7449.863,E2 -7449.863} C_VEL
LIN {X 0,Y 471.211,Z 336.788,A -85,B 0,C 180,E1 -7451.014,E2 -7451.014} C_VEL
LIN {X 0,Y 468.746,Z 337.096,A -85,B 0,C 180,E1 -7451.941,E2 -7451.941} C_VEL
LIN {X 0,Y 467.679,Z 337.228,A -85,B 0,C 180,E1 -7452.659,E2 -7452.659} C_VEL
LIN {X 0,Y 467.591,Z 337.238,A -85,B 0,C 180,E1 -7452.902,E2 -7452.902} C_VEL
LIN {X 0,Y 467.608,Z 337.237,A -85,B 0,C 180,E1 -7455.196,E2 -7455.196} C_VEL
LIN {X 0,Y 467.657,Z 337.233,A -85,B 0,C 180,E1 -7457.855,E2 -7457.855} C_VEL
LIN {X 0,Y 467.683,Z 337.23,A -85,B 0,C 180,E1 -7461.357,E2 -7461.357} C_VEL
LIN {X 0,Y 467.737,Z 337.221,A -85,B 0,C 180,E1 -7463.963,E2 -7463.963} C_VEL
LIN {X 0,Y 467.861,Z 337.204,A -85,B 0,C 180,E1 -7467.417,E2 -7467.417} C_VEL
LIN {X 0,Y 467.884,Z 337.206,A -85,B 0,C 180,E1 -7470,E2 -7470} C_VEL
LIN {X 0,Y 467.862,Z 337.204,A -85,B 0,C 180,E1 -7472.583,E2 -7472.583} C_VEL
LIN {X 0,Y 467.737,Z 337.221,A -85,B 0,C 180,E1 -7476.038,E2 -7476.038} C_VEL
LIN {X 0,Y 467.684,Z 337.229,A -85,B 0,C 180,E1 -7478.643,E2 -7478.643} C_VEL
LIN {X 0,Y 467.658,Z 337.235,A -85,B 0,C 180,E1 -7482.146,E2 -7482.146} C_VEL
LIN {X 0,Y 467.641,Z 337.236,A -85,B 0,C 180,E1 -7485.695,E2 -7485.695} C_VEL
LIN {X 0,Y 467.619,Z 337.235,A -85,B 0,C 180,E1 -7488.765,E2 -7488.765} C_VEL
LIN {X 0,Y 467.582,Z 337.244,A -85,B 0,C 180,E1 -7491.268,E2 -7491.268} C_VEL
LIN {X 0,Y 467.574,Z 337.241,A -85,B 0,C 180,E1 -7493.944,E2 -7493.944} C_VEL
LIN {X 0,Y 467.618,Z 337.238,A -85,B 0,C 180,E1 -7496.8,E2 -7496.8} C_VEL
LIN {X 0,Y 467.556,Z 337.247,A -85,B 0,C 180,E1 -7499.738,E2 -7499.738} C_VEL
LIN {X 0,Y 467.585,Z 337.238,A -85,B 0,C 180,E1 -7502.759,E2 -7502.759} C_VEL
LIN {X 0,Y 467.555,Z 337.243,A -85,B 0,C 180,E1 -7505.89,E2 -7505.89} C_VEL
LIN {X 0,Y 467.584,Z 337.242,A -85,B 0,C 180,E1 -7509.145,E2 -7509.145} C_VEL
LIN {X 0,Y 467.622,Z 337.238,A -85,B 0,C 180,E1 -7512.572,E2 -7512.572} C_VEL
LIN {X 0,Y 467.573,Z 337.241,A -85,B 0,C 180,E1 -7515.054,E2 -7515.054} C_VEL
LIN {X 0,Y 467.591,Z 337.242,A -85,B 0,C 180,E1 -7517.44,E2 -7517.44} C_VEL
LIN {X 0,Y 467.585,Z 337.24,A -85,B 0,C 180,E1 -7520.856,E2 -7520.856} C_VEL
LIN {X 0,Y 467.564,Z 337.242,A -85,B 0,C 180,E1 -7524.261,E2 -7524.261} C_VEL
LIN {X 0,Y 467.585,Z 337.24,A -85,B 0,C 180,E1 -7527.321,E2 -7527.321} C_VEL
LIN {X 0,Y 467.574,Z 337.242,A -85,B 0,C 180,E1 -7530.668,E2 -7530.668} C_VEL
LIN {X 0,Y 467.621,Z 337.237,A -85,B 0,C 180,E1 -7533.2,E2 -7533.2} C_VEL
LIN {X 0,Y 467.597,Z 337.238,A -85,B 0,C 180,E1 -7536.469,E2 -7536.469} C_VEL
LIN {X 0,Y 467.627,Z 337.232,A -85,B 0,C 180,E1 -7539.777,E2 -7539.777} C_VEL
LIN {X 0,Y 467.611,Z 337.24,A -85,B 0,C 180,E1 -7542.507,E2 -7542.507} C_VEL
LIN {X 0,Y 467.612,Z 337.236,A -85,B 0,C 180,E1 -7545.197,E2 -7545.197} C_VEL
LIN {X 0,Y 467.662,Z 337.232,A -85,B 0,C 180,E1 -7547.855,E2 -7547.855} C_VEL
LIN {X 0,Y 467.688,Z 337.229,A -85,B 0,C 180,E1 -7551.357,E2 -7551.357} C_VEL
LIN {X 0,Y 467.749,Z 337.218,A -85,B 0,C 180,E1 -7553.963,E2 -7553.963} C_VEL
LIN {X 0,Y 467.863,Z 337.203,A -85,B 0,C 180,E1 -7557.417,E2 -7557.417} C_VEL
LIN {X 0,Y 467.888,Z 337.203,A -85,B 0,C 180,E1 -7560,E2 -7560} C_VEL
LIN {X 0,Y 467.865,Z 337.205,A -85,B 0,C 180,E1 -7562.583,E2 -7562.583} C_VEL
LIN {X 0,Y 467.739,Z 337.222,A -85,B 0,C 180,E1 -7566.038,E2 -7566.038} C_VEL
LIN {X 0,Y 467.675,Z 337.231,A -85,B 0,C 180,E1 -7568.643,E2 -7568.643} C_VEL
LIN {X 0,Y 467.662,Z 337.231,A -85,B 0,C 180,E1 -7572.145,E2 -7572.145} C_VEL
LIN {X 0,Y 467.645,Z 337.232,A -85,B 0,C 180,E1 -7575.695,E2 -7575.695} C_VEL
LIN {X 0,Y 467.624,Z 337.234,A -85,B 0,C 180,E1 -7578.765,E2 -7578.765} C_VEL
LIN {X 0,Y 467.586,Z 337.241,A -85,B 0,C 180,E1 -7581.268,E2 -7581.268} C_VEL
LIN {X 0,Y 467.577,Z 337.241,A -85,B 0,C 180,E1 -7583.943,E2 -7583.943} C_VEL
LIN {X 0,Y 467.622,Z 337.237,A -85,B 0,C 180,E1 -7586.8,E2 -7586.8} C_VEL
LIN {X 0,Y 467.559,Z 337.243,A -85,B 0,C 180,E1 -7589.738,E2 -7589.738} C_VEL
LIN {X 0,Y 467.588,Z 337.237,A -85,B 0,C 180,E1 -7592.758,E2 -7592.758} C_VEL
LIN {X 0,Y 467.561,Z 337.245,A -85,B 0,C 180,E1 -7595.889,E2 -7595.889} C_VEL
LIN {X 0,Y 467.587,Z 337.242,A -85,B 0,C 180,E1 -7599.144,E2 -7599.144} C_VEL
LIN {X 0,Y 467.591,Z 337.243,A -85,B 0,C 180,E1 -7602.567,E2 -7602.567} C_VEL
LIN {X 0,Y 467.575,Z 337.242,A -85,B 0,C 180,E1 -7605.053,E2 -7605.053} C_VEL
LIN {X 0,Y 467.593,Z 337.24,A -85,B 0,C 180,E1 -7607.44,E2 -7607.44} C_VEL
LIN {X 0,Y 467.609,Z 337.379,A -85,B 0,C 180,E1 -7609.029,E2 -7609.029} C_VEL
LIN {X 0,Y 469.813,Z 348.297,A -85,B 0,C 180,E1 -7612.169,E2 -7612.169} C_VEL
LIN {X 0,Y 470.611,Z 354.07,A -85,B 0,C 180,E1 -7613.748,E2 -7613.748} C_VEL
LIN {X 0,Y 469.85,Z 366.422,A -85,B 0,C 180,E1 -7616.893,E2 -7616.893} C_VEL
LIN {X 0,Y 469.302,Z 377.504,A -85,B 0,C 180,E1 -7619.641,E2 -7619.641} C_VEL
LIN {X 0,Y 468.794,Z 390.501,A -85,B 0,C 180,E1 -7622.79,E2 -7622.79} C_VEL
LIN {X 0,Y 468.235,Z 405.262,A -85,B 0,C 180,E1 -7626.289,E2 -7626.289} C_VEL
LIN {X 0,Y 467.765,Z 420.323,A -85,B 0,C 180,E1 -7629.783,E2 -7629.783} C_VEL
LIN {X 0,Y 467.469,Z 432.2,A -85,B 0,C 180,E1 -7632.501,E2 -7632.501} C_VEL
LIN {X 0,Y 467.278,Z 441.447,A -85,B 0,C 180,E1 -7634.6,E2 -7634.6} C_VEL
LIN {X 0,Y 468.765,Z 457.359,A -85,B 0,C 180,E1 -7635.081,E2 -7635.081} C_VEL
LIN {X 0,Y 469.639,Z 465.622,A -85,B 0,C 180,E1 -7635.428,E2 -7635.428} C_VEL
LIN {X 0,Y 469.141,Z 477.607,A -85,B 0,C 180,E1 -7636.021,E2 -7636.021} C_VEL
LIN {X 0,Y 468.643,Z 489.377,A -85,B 0,C 180,E1 -7636.779,E2 -7636.779} C_VEL
LIN {X 0,Y 468.218,Z 500.942,A -85,B 0,C 180,E1 -7637.733,E2 -7637.733} C_VEL
LIN {X 0,Y 467.731,Z 510.797,A -85,B 0,C 180,E1 -7638.736,E2 -7638.736} C_VEL
LIN {X 0,Y 467.387,Z 519.589,A -85,B 0,C 180,E1 -7639.823,E2 -7639.823} C_VEL
LIN {X 0,Y 467.118,Z 528.157,A -85,B 0,C 180,E1 -7641.129,E2 -7641.129} C_VEL
LIN {X 0,Y 467.007,Z 535.055,A -85,B 0,C 180,E1 -7642.433,E2 -7642.433} C_VEL
LIN {X 0,Y 466.999,Z 541.39,A -85,B 0,C 180,E1 -7643.953,E2 -7643.953} C_VEL
LIN {X 0,Y 466.944,Z 545.478,A -85,B 0,C 180,E1 -7645.251,E2 -7645.251} C_VEL
LIN {X 0,Y 466.962,Z 548.481,A -85,B 0,C 180,E1 -7646.549,E2 -7646.549} C_VEL
LIN {X 0,Y 466.948,Z 549.908,A -85,B 0,C 180,E1 -7647.412,E2 -7647.412} C_VEL
LIN {X 0,Y 466.935,Z 550.895,A -85,B 0,C 180,E1 -7648.275,E2 -7648.275} C_VEL
LIN {X 0,Y 467.059,Z 551.662,A -85,B 0,C 180,E1 -7650,E2 -7650} C_VEL
LIN {X 0,Y 467.077,Z 551.379,A -85,B 0,C 180,E1 -7650.862,E2 -7650.862} C_VEL
LIN {X 0,Y 466.993,Z 549.539,A -85,B 0,C 180,E1 -7652.588,E2 -7652.588} C_VEL
LIN {X 0,Y 467.045,Z 547.022,A -85,B 0,C 180,E1 -7653.883,E2 -7653.883} C_VEL
LIN {X 0,Y 467.038,Z 543.443,A -85,B 0,C 180,E1 -7655.18,E2 -7655.18} C_VEL
LIN {X 0,Y 467.055,Z 537.758,A -85,B 0,C 180,E1 -7656.716,E2 -7656.716} C_VEL
LIN {X 0,Y 467.15,Z 530.421,A -85,B 0,C 180,E1 -7658.217,E2 -7658.217} C_VEL
LIN {X 0,Y 467.298,Z 522.431,A -85,B 0,C 180,E1 -7659.523,E2 -7659.523} C_VEL
LIN {X 0,Y 467.535,Z 514.318,A -85,B 0,C 180,E1 -7660.611,E2 -7660.611} C_VEL
LIN {X 0,Y 467.885,Z 504.48,A -85,B 0,C 180,E1 -7661.7,E2 -7661.7} C_VEL
LIN {X 0,Y 468.222,Z 493.785,A -85,B 0,C 180,E1 -7662.669,E2 -7662.669} C_VEL
LIN {X 0,Y 468.742,Z 481.803,A -85,B 0,C 180,E1 -7663.549,E2 -7663.549} C_VEL
LIN {X 0,Y 469.238,Z 469.476,A -85,B 0,C 180,E1 -7664.252,E2 -7664.252} C_VEL
LIN {X 0,Y 469.309,Z 463.683,A -85,B 0,C 180,E1 -7664.527,E2 -7664.527} C_VEL
LIN {X 0,Y 468.407,Z 453.861,A -85,B 0,C 180,E1 -7664.944,E2 -7664.944} C_VEL
LIN {X 0,Y 467.415,Z 439.27,A -85,B 0,C 180,E1 -7665.385,E2 -7665.385} C_VEL
LIN {X 0,Y 467.27,Z 437.291,A -85,B 0,C 180,E1 -7665.456,E2 -7665.456} C_VEL
LIN {X 0,Y 467.43,Z 423.51,A -85,B 0,C 180,E1 -7668.406,E2 -7668.406} C_VEL
LIN {X 0,Y 467.563,Z 410.307,A -85,B 0,C 180,E1 -7671.262,E2 -7671.262} C_VEL
LIN {X 0,Y 467.776,Z 396.056,A -85,B 0,C 180,E1 -7674.404,E2 -7674.404} C_VEL
LIN {X 0,Y 468.013,Z 383.709,A -85,B 0,C 180,E1 -7677.204,E2 -7677.204} C_VEL
LIN {X 0,Y 468.289,Z 371.09,A -85,B 0,C 180,E1 -7680.183,E2 -7680.183} C_VEL
LIN {X 0,Y 468.674,Z 360.226,A -85,B 0,C 180,E1 -7682.886,E2 -7682.886} C_VEL
LIN {X 0,Y 469.504,Z 348.343,A -85,B 0,C 180,E1 -7686.067,E2 -7686.067} C_VEL
LIN {X 0,Y 468.917,Z 343.98,A -85,B 0,C 180,E1 -7687.406,E2 -7687.406} C_VEL
LIN {X 0,Y 467.586,Z 337.245,A -85,B 0,C 180,E1 -7689.747,E2 -7689.747} C_VEL
LIN {X 0,Y 467.59,Z 337.242,A -85,B 0,C 180,E1 -7692.567,E2 -7692.567} C_VEL
LIN {X 0,Y 467.574,Z 337.244,A -85,B 0,C 180,E1 -7695.053,E2 -7695.053} C_VEL
LIN {X 0,Y 467.592,Z 337.242,A -85,B 0,C 180,E1 -7697.44,E2 -7697.44} C_VEL
LIN {X 0,Y 467.586,Z 337.24,A -85,B 0,C 180,E1 -7700.855,E2 -7700.855} C_VEL
LIN {X 0,Y 467.566,Z 337.245,A -85,B 0,C 180,E1 -7704.26,E2 -7704.26} C_VEL
LIN {X 0,Y 467.586,Z 337.242,A -85,B 0,C 180,E1 -7707.321,E2 -7707.321} C_VEL
LIN {X 0,Y 467.574,Z 337.241,A -85,B 0,C 180,E1 -7710.667,E2 -7710.667} C_VEL
LIN {X 0,Y 467.617,Z 337.236,A -85,B 0,C 180,E1 -7713.2,E2 -7713.2} C_VEL
LIN {X 0,Y 467.595,Z 337.24,A -85,B 0,C 180,E1 -7716.469,E2 -7716.469} C_VEL
LIN {X 0,Y 467.627,Z 337.238,A -85,B 0,C 180,E1 -7719.777,E2 -7719.777} C_VEL
LIN {X 0,Y 467.611,Z 337.24,A -85,B 0,C 180,E1 -7722.507,E2 -7722.507} C_VEL
LIN {X 0,Y 467.656,Z 337.26,A -85,B 0,C 180,E1 -7724.403,E2 -7724.403} C_VEL
LIN {X 0,Y 470.441,Z 347.48,A -85,B 0,C 180,E1 -7725.066,E2 -7725.066} C_VEL
LIN {X 0,Y 470.079,Z 359.012,A -85,B 0,C 180,E1 -7725.829,E2 -7725.829} C_VEL
LIN {X 0,Y 469.729,Z 368.933,A -85,B 0,C 180,E1 -7726.65,E2 -7726.65} C_VEL
LIN {X 0,Y 469.289,Z 378.962,A -85,B 0,C 180,E1 -7727.678,E2 -7727.678} C_VEL
LIN {X 0,Y 468.831,Z 387.594,A -85,B 0,C 180,E1 -7728.762,E2 -7728.762} C_VEL
LIN {X 0,Y 468.445,Z 395.985,A -85,B 0,C 180,E1 -7730.065,E2 -7730.065} C_VEL
LIN {X 0,Y 468.106,Z 402.641,A -85,B 0,C 180,E1 -7731.365,E2 -7731.365} C_VEL
LIN {X 0,Y 467.817,Z 407.476,A -85,B 0,C 180,E1 -7732.534,E2 -7732.534} C_VEL
LIN {X 0,Y 467.697,Z 412.018,A -85,B 0,C 180,E1 -7733.962,E2 -7733.962} C_VEL
LIN {X 0,Y 467.458,Z 414.184,A -85,B 0,C 180,E1 -7734.824,E2 -7734.824} C_VEL
LIN {X 0,Y 467.388,Z 415.896,A -85,B 0,C 180,E1 -7735.688,E2 -7735.688} C_VEL
LIN {X 0,Y 467.322,Z 417.146,A -85,B 0,C 180,E1 -7736.551,E2 -7736.551} C_VEL
LIN {X 0,Y 467.251,Z 418.481,A -85,B 0,C 180,E1 -7738.276,E2 -7738.276} C_VEL
LIN {X 0,Y 467.181,Z 418.56,A -85,B 0,C 180,E1 -7739.138,E2 -7739.138} C_VEL
LIN {X 0,Y 467.184,Z 417.474,A -85,B 0,C 180,E1 -7740.862,E2 -7740.862} C_VEL
LIN {X 0,Y 467.255,Z 416.348,A -85,B 0,C 180,E1 -7741.724,E2 -7741.724} C_VEL
LIN {X 0,Y 467.288,Z 413.864,A -85,B 0,C 180,E1 -7743.017,E2 -7743.017} C_VEL
LIN {X 0,Y 467.438,Z 410.385,A -85,B 0,C 180,E1 -7744.311,E2 -7744.311} C_VEL
LIN {X 0,Y 467.598,Z 405.833,A -85,B 0,C 180,E1 -7745.606,E2 -7745.606} C_VEL
LIN {X 0,Y 467.961,Z 400.05,A -85,B 0,C 180,E1 -7746.9,E2 -7746.9} C_VEL
LIN {X 0,Y 468.209,Z 392.837,A -85,B 0,C 180,E1 -7748.198,E2 -7748.198} C_VEL
LIN {X 0,Y 468.585,Z 383.875,A -85,B 0,C 180,E1 -7749.496,E2 -7749.496} C_VEL
LIN {X 0,Y 469.016,Z 374.681,A -85,B 0,C 180,E1 -7750.577,E2 -7750.577} C_VEL
LIN {X 0,Y 469.418,Z 364.482,A -85,B 0,C 180,E1 -7751.551,E2 -7751.551} C_VEL
LIN {X 0,Y 469.688,Z 355.524,A -85,B 0,C 180,E1 -7752.261,E2 -7752.261} C_VEL
LIN {X 0,Y 470.026,Z 346.376,A -85,B 0,C 180,E1 -7752.859,E2 -7752.859} C_VEL
LIN {X 0,Y 467.616,Z 337.239,A -85,B 0,C 180,E1 -7753.457,E2 -7753.457} C_VEL
LIN {X 0,Y 467.595,Z 337.237,A -85,B 0,C 180,E1 -7756.593,E2 -7756.593} C_VEL
LIN {X 0,Y 467.625,Z 337.237,A -85,B 0,C 180,E1 -7759.308,E2 -7759.308} C_VEL
LIN {X 0,Y 467.538,Z 337.246,A -85,B 0,C 180,E1 -7762.074,E2 -7762.074} C_VEL
LIN {X 0,Y 467.606,Z 337.239,A -85,B 0,C 180,E1 -7764.887,E2 -7764.887} C_VEL
LIN {X 0,Y 467.631,Z 337.236,A -85,B 0,C 180,E1 -7767.768,E2 -7767.768} C_VEL
LIN {X 0,Y 467.572,Z 337.243,A -85,B 0,C 180,E1 -7771.045,E2 -7771.045} C_VEL
LIN {X 0,Y 467.591,Z 337.237,A -85,B 0,C 180,E1 -7774.242,E2 -7774.242} C_VEL
LIN {X 0,Y 467.551,Z 337.244,A -85,B 0,C 180,E1 -7777.186,E2 -7777.186} C_VEL
